    CONST robtarget p15959:= [[1433.0986274492811, 9.608746814305746, 1008.500033578516], [0, 0, 1, 0], [0, 0, 0, 0], [9E9, 9E9, 9E9, 9E9, 9E9, 9E9]];
    CONST robtarget p15960:= [[1433.1589710304575, 10.015424002704279, 1008.500033578516], [0, 0, 1, 0], [0, 0, 0, 0], [9E9, 9E9, 9E9, 9E9, 9E9, 9E9]];
    CONST robtarget p15961:= [[1433.2058201782734, 10.459822262926878, 1008.500033578516], [0, 0, 1, 0], [0, 0, 0, 0], [9E9, 9E9, 9E9, 9E9, 9E9, 9E9]];
    CONST robtarget p15962:= [[1433.4130381026719, 11.206085604370102, 1008.500033578516], [0, 0, 1, 0], [0, 0, 0, 0], [9E9, 9E9, 9E9, 9E9, 9E9, 9E9]];
    CONST robtarget p15963:= [[1433.6247056823859, 12.59383709002276, 1008.500033578516], [0, 0, 1, 0], [0, 0, 0, 0], [9E9, 9E9, 9E9, 9E9, 9E9, 9E9]];
    CONST robtarget p15964:= [[1433.6430735052686, 12.762150805315983, 1008.500033578516], [0, 0, 1, 0], [0, 0, 0, 0], [9E9, 9E9, 9E9, 9E9, 9E9, 9E9]];
    CONST robtarget p15965:= [[1433.7465034826027, 13.275407559875234, 1008.500033578516], [0, 0, 1, 0], [0, 0, 0, 0], [9E9, 9E9, 9E9, 9E9, 9E9, 9E9]];
    CONST robtarget p15966:= [[1433.7741777327235, 13.488161726566162, 1008.500033578516], [0, 0, 1, 0], [0, 0, 0, 0], [9E9, 9E9, 9E9, 9E9, 9E9, 9E9]];
    CONST robtarget p15967:= [[1433.8795125581278, 13.879378212952375, 1008.500033578516], [0, 0, 1, 0], [0, 0, 0, 0], [9E9, 9E9, 9E9, 9E9, 9E9, 9E9]];
    CONST robtarget p15968:= [[1433.9684930832368, 14.246080535111645, 1008.500033578516], [0, 0, 1, 0], [0, 0, 0, 0], [9E9, 9E9, 9E9, 9E9, 9E9, 9E9]];
    CONST robtarget p15969:= [[1434.0660993207537, 14.620211943199038, 1008.500033578516], [0, 0, 1, 0], [0, 0, 0, 0], [9E9, 9E9, 9E9, 9E9, 9E9, 9E9]];
    CONST robtarget p15970:= [[1434.095837116519, 14.758515891180053, 1008.500033578516], [0, 0, 1, 0], [0, 0, 0, 0], [9E9, 9E9, 9E9, 9E9, 9E9, 9E9]];
    CONST robtarget p15971:= [[1434.245693850769, 15.479233166590063, 1008.500033578516], [0, 0, 1, 0], [0, 0, 0, 0], [9E9, 9E9, 9E9, 9E9, 9E9, 9E9]];
    CONST robtarget p15972:= [[1434.4221561340992, 16.325849023968487, 1008.500033578516], [0, 0, 1, 0], [0, 0, 0, 0], [9E9, 9E9, 9E9, 9E9, 9E9, 9E9]];
    CONST robtarget p15973:= [[1434.61472670305, 16.937455427209215, 1008.500033578516], [0, 0, 1, 0], [0, 0, 0, 0], [9E9, 9E9, 9E9, 9E9, 9E9, 9E9]];
    CONST robtarget p15974:= [[1434.7025719249725, 17.322639850120922, 1008.500033578516], [0, 0, 1, 0], [0, 0, 0, 0], [9E9, 9E9, 9E9, 9E9, 9E9, 9E9]];
    CONST robtarget p15975:= [[1434.9090055185184, 18.0090372974757, 1008.500033578516], [0, 0, 1, 0], [0, 0, 0, 0], [9E9, 9E9, 9E9, 9E9, 9E9, 9E9]];
    CONST robtarget p15976:= [[1435.0307135396993, 18.599825888870924, 1008.500033578516], [0, 0, 1, 0], [0, 0, 0, 0], [9E9, 9E9, 9E9, 9E9, 9E9, 9E9]];
    CONST robtarget p15977:= [[1435.0769349823054, 18.84950465909236, 1008.500033578516], [0, 0, 1, 0], [0, 0, 0, 0], [9E9, 9E9, 9E9, 9E9, 9E9, 9E9]];
    CONST robtarget p15978:= [[1435.1457068870573, 19.06963509468285, 1008.500033578516], [0, 0, 1, 0], [0, 0, 0, 0], [9E9, 9E9, 9E9, 9E9, 9E9, 9E9]];
    CONST robtarget p15979:= [[1435.2539630872568, 19.45271986997699, 1008.500033578516], [0, 0, 1, 0], [0, 0, 0, 0], [9E9, 9E9, 9E9, 9E9, 9E9, 9E9]];
    CONST robtarget p15980:= [[1435.2779629825206, 19.54379334494176, 1008.500033578516], [0, 0, 1, 0], [0, 0, 0, 0], [9E9, 9E9, 9E9, 9E9, 9E9, 9E9]];
    CONST robtarget p15981:= [[1435.30275284433, 19.612075769745374, 1008.500033578516], [0, 0, 1, 0], [0, 0, 0, 0], [9E9, 9E9, 9E9, 9E9, 9E9, 9E9]];
    CONST robtarget p15982:= [[1435.4854707109937, 20.199981390981975, 1008.500033578516], [0, 0, 1, 0], [0, 0, 0, 0], [9E9, 9E9, 9E9, 9E9, 9E9, 9E9]];
    CONST robtarget p15983:= [[1435.5853392667057, 20.482104936748172, 1008.500033578516], [0, 0, 1, 0], [0, 0, 0, 0], [9E9, 9E9, 9E9, 9E9, 9E9, 9E9]];
    CONST robtarget p15984:= [[1435.7681134476982, 21.021407578977716, 1008.500033578516], [0, 0, 1, 0], [0, 0, 0, 0], [9E9, 9E9, 9E9, 9E9, 9E9, 9E9]];
    CONST robtarget p15985:= [[1435.958175713581, 21.47955589963057, 1008.500033578516], [0, 0, 1, 0], [0, 0, 0, 0], [9E9, 9E9, 9E9, 9E9, 9E9, 9E9]];
    CONST robtarget p15986:= [[1436.1023198224916, 21.945686573091862, 1008.500033578516], [0, 0, 1, 0], [0, 0, 0, 0], [9E9, 9E9, 9E9, 9E9, 9E9, 9E9]];
    CONST robtarget p15987:= [[1436.1825943607196, 22.203311510029366, 1008.500033578516], [0, 0, 1, 0], [0, 0, 0, 0], [9E9, 9E9, 9E9, 9E9, 9E9, 9E9]];
    CONST robtarget p15988:= [[1436.349538758373, 22.703386458321205, 1008.500033578516], [0, 0, 1, 0], [0, 0, 0, 0], [9E9, 9E9, 9E9, 9E9, 9E9, 9E9]];
    CONST robtarget p15989:= [[1436.6119112199715, 23.432726370190338, 1008.500033578516], [0, 0, 1, 0], [0, 0, 0, 0], [9E9, 9E9, 9E9, 9E9, 9E9, 9E9]];
    CONST robtarget p15990:= [[1436.7778943099147, 23.981953823344938, 1008.500033578516], [0, 0, 1, 0], [0, 0, 0, 0], [9E9, 9E9, 9E9, 9E9, 9E9, 9E9]];
    CONST robtarget p15991:= [[1437.0642227941967, 24.65637773782116, 1008.500033578516], [0, 0, 1, 0], [0, 0, 0, 0], [9E9, 9E9, 9E9, 9E9, 9E9, 9E9]];
    CONST robtarget p15992:= [[1437.2587373872966, 25.12385144143589, 1008.500033578516], [0, 0, 1, 0], [0, 0, 0, 0], [9E9, 9E9, 9E9, 9E9, 9E9, 9E9]];
    CONST robtarget p15993:= [[1437.3936146926897, 25.408671993782846, 1008.500033578516], [0, 0, 1, 0], [0, 0, 0, 0], [9E9, 9E9, 9E9, 9E9, 9E9, 9E9]];
    CONST robtarget p15994:= [[1437.6905856905832, 26.057288547637995, 1008.500033578516], [0, 0, 1, 0], [0, 0, 0, 0], [9E9, 9E9, 9E9, 9E9, 9E9, 9E9]];
    CONST robtarget p15995:= [[1437.8323968402112, 26.419387210097497, 1008.500033578516], [0, 0, 1, 0], [0, 0, 0, 0], [9E9, 9E9, 9E9, 9E9, 9E9, 9E9]];
    CONST robtarget p15996:= [[1437.954968895154, 26.72409400055281, 1008.500033578516], [0, 0, 1, 0], [0, 0, 0, 0], [9E9, 9E9, 9E9, 9E9, 9E9, 9E9]];
    CONST robtarget p15997:= [[1438.0143479796734, 26.878363265785197, 1008.500033578516], [0, 0, 1, 0], [0, 0, 0, 0], [9E9, 9E9, 9E9, 9E9, 9E9, 9E9]];
    CONST robtarget p15998:= [[1438.0697366851261, 27.02314795976943, 1008.500033578516], [0, 0, 1, 0], [0, 0, 0, 0], [9E9, 9E9, 9E9, 9E9, 9E9, 9E9]];
    CONST robtarget p15999:= [[1438.2271993834418, 27.43282297537347, 1008.500033578516], [0, 0, 1, 0], [0, 0, 0, 0], [9E9, 9E9, 9E9, 9E9, 9E9, 9E9]];
    CONST robtarget p16000:= [[1438.4463940522078, 27.84677822927749, 1008.500033578516], [0, 0, 1, 0], [0, 0, 0, 0], [9E9, 9E9, 9E9, 9E9, 9E9, 9E9]];
    CONST robtarget p16001:= [[1438.7558501610374, 28.663010257655827, 1008.500033578516], [0, 0, 1, 0], [0, 0, 0, 0], [9E9, 9E9, 9E9, 9E9, 9E9, 9E9]];
    CONST robtarget p16002:= [[1438.9070799315605, 28.90804462441197, 1008.500033578516], [0, 0, 1, 0], [0, 0, 0, 0], [9E9, 9E9, 9E9, 9E9, 9E9, 9E9]];
    CONST robtarget p16003:= [[1439.2433018788113, 29.59362072222892, 1008.500033578516], [0, 0, 1, 0], [0, 0, 0, 0], [9E9, 9E9, 9E9, 9E9, 9E9, 9E9]];
    CONST robtarget p16004:= [[1439.4746197403977, 30.0450442591478, 1008.500033578516], [0, 0, 1, 0], [0, 0, 0, 0], [9E9, 9E9, 9E9, 9E9, 9E9, 9E9]];
    CONST robtarget p16005:= [[1439.7668782569137, 30.57529808046486, 1008.500033578516], [0, 0, 1, 0], [0, 0, 0, 0], [9E9, 9E9, 9E9, 9E9, 9E9, 9E9]];
    CONST robtarget p16006:= [[1440.177882853498, 31.2929706114746, 1008.500033578516], [0, 0, 1, 0], [0, 0, 0, 0], [9E9, 9E9, 9E9, 9E9, 9E9, 9E9]];
    CONST robtarget p16007:= [[1440.5677510154408, 32.1772795548887, 1008.500033578516], [0, 0, 1, 0], [0, 0, 0, 0], [9E9, 9E9, 9E9, 9E9, 9E9, 9E9]];
    CONST robtarget p16008:= [[1440.9506297367848, 32.90687188456482, 1008.500033578516], [0, 0, 1, 0], [0, 0, 0, 0], [9E9, 9E9, 9E9, 9E9, 9E9, 9E9]];
    CONST robtarget p16009:= [[1441.0515934210391, 33.082825334749856, 1008.500033578516], [0, 0, 1, 0], [0, 0, 0, 0], [9E9, 9E9, 9E9, 9E9, 9E9, 9E9]];
    CONST robtarget p16010:= [[1441.291561344643, 33.51277826861488, 1008.500033578516], [0, 0, 1, 0], [0, 0, 0, 0], [9E9, 9E9, 9E9, 9E9, 9E9, 9E9]];
    CONST robtarget p16011:= [[1441.4170597081568, 33.71755199461752, 1008.500033578516], [0, 0, 1, 0], [0, 0, 0, 0], [9E9, 9E9, 9E9, 9E9, 9E9, 9E9]];
    CONST robtarget p16012:= [[1441.6717736369376, 34.087403365805486, 1008.500033578516], [0, 0, 1, 0], [0, 0, 0, 0], [9E9, 9E9, 9E9, 9E9, 9E9, 9E9]];
    CONST robtarget p16013:= [[1442.0183475741433, 34.67340426693394, 1008.500033578516], [0, 0, 1, 0], [0, 0, 0, 0], [9E9, 9E9, 9E9, 9E9, 9E9, 9E9]];
    CONST robtarget p16014:= [[1442.1305600956955, 34.842443823146525, 1008.500033578516], [0, 0, 1, 0], [0, 0, 0, 0], [9E9, 9E9, 9E9, 9E9, 9E9, 9E9]];
    CONST robtarget p16015:= [[1442.8215804591978, 35.99192933058819, 1008.500033578516], [0, 0, 1, 0], [0, 0, 0, 0], [9E9, 9E9, 9E9, 9E9, 9E9, 9E9]];
    CONST robtarget p16016:= [[1443.1406638568508, 36.489162717446646, 1008.500033578516], [0, 0, 1, 0], [0, 0, 0, 0], [9E9, 9E9, 9E9, 9E9, 9E9, 9E9]];
    CONST robtarget p16017:= [[1443.254415228456, 36.68748397793732, 1008.500033578516], [0, 0, 1, 0], [0, 0, 0, 0], [9E9, 9E9, 9E9, 9E9, 9E9, 9E9]];
    CONST robtarget p16018:= [[1443.4510665943017, 37.071600292545924, 1008.500033578516], [0, 0, 1, 0], [0, 0, 0, 0], [9E9, 9E9, 9E9, 9E9, 9E9, 9E9]];
    CONST robtarget p16019:= [[1443.9592495899064, 37.76667396099968, 1008.500033578516], [0, 0, 1, 0], [0, 0, 0, 0], [9E9, 9E9, 9E9, 9E9, 9E9, 9E9]];
    CONST robtarget p16020:= [[1444.4069080527252, 38.4188532456172, 1008.500033578516], [0, 0, 1, 0], [0, 0, 0, 0], [9E9, 9E9, 9E9, 9E9, 9E9, 9E9]];
    CONST robtarget p16021:= [[1444.7601463802437, 38.874871104904, 1008.500033578516], [0, 0, 1, 0], [0, 0, 0, 0], [9E9, 9E9, 9E9, 9E9, 9E9, 9E9]];
    CONST robtarget p16022:= [[1445.248558127412, 39.600155696272054, 1008.500033578516], [0, 0, 1, 0], [0, 0, 0, 0], [9E9, 9E9, 9E9, 9E9, 9E9, 9E9]];
    CONST robtarget p16023:= [[1445.294443015287, 39.67172478622983, 1008.500033578516], [0, 0, 1, 0], [0, 0, 0, 0], [9E9, 9E9, 9E9, 9E9, 9E9, 9E9]];
    CONST robtarget p16024:= [[1445.3797142458502, 39.77745344396661, 1008.500033578516], [0, 0, 1, 0], [0, 0, 0, 0], [9E9, 9E9, 9E9, 9E9, 9E9, 9E9]];
    CONST robtarget p16025:= [[1445.7587485571103, 40.28723104743635, 1008.500033578516], [0, 0, 1, 0], [0, 0, 0, 0], [9E9, 9E9, 9E9, 9E9, 9E9, 9E9]];
    CONST robtarget p16026:= [[1446.01804192666, 40.63892152668981, 1008.500033578516], [0, 0, 1, 0], [0, 0, 0, 0], [9E9, 9E9, 9E9, 9E9, 9E9, 9E9]];
    CONST robtarget p16027:= [[1446.312375477045, 41.03187796392518, 1008.500033578516], [0, 0, 1, 0], [0, 0, 0, 0], [9E9, 9E9, 9E9, 9E9, 9E9, 9E9]];
    CONST robtarget p16028:= [[1446.4254911527705, 41.16274682131454, 1008.500033578516], [0, 0, 1, 0], [0, 0, 0, 0], [9E9, 9E9, 9E9, 9E9, 9E9, 9E9]];
    CONST robtarget p16029:= [[1446.9971446431318, 41.842211595922834, 1008.500033578516], [0, 0, 1, 0], [0, 0, 0, 0], [9E9, 9E9, 9E9, 9E9, 9E9, 9E9]];
    CONST robtarget p16030:= [[1447.3278104158244, 42.321049762311645, 1008.500033578516], [0, 0, 1, 0], [0, 0, 0, 0], [9E9, 9E9, 9E9, 9E9, 9E9, 9E9]];
    CONST robtarget p16031:= [[1447.6388954335016, 42.65857624043116, 1008.500033578516], [0, 0, 1, 0], [0, 0, 0, 0], [9E9, 9E9, 9E9, 9E9, 9E9, 9E9]];
    CONST robtarget p16032:= [[1448.0381842833888, 43.178669383244966, 1008.500033578516], [0, 0, 1, 0], [0, 0, 0, 0], [9E9, 9E9, 9E9, 9E9, 9E9, 9E9]];
    CONST robtarget p16033:= [[1448.366752181317, 43.60401220044736, 1008.500033578516], [0, 0, 1, 0], [0, 0, 0, 0], [9E9, 9E9, 9E9, 9E9, 9E9, 9E9]];
    CONST robtarget p16034:= [[1448.5125298028045, 43.76454658599833, 1008.500033578516], [0, 0, 1, 0], [0, 0, 0, 0], [9E9, 9E9, 9E9, 9E9, 9E9, 9E9]];
    CONST robtarget p16035:= [[1448.7672952912585, 44.07132722933555, 1008.500033578516], [0, 0, 1, 0], [0, 0, 0, 0], [9E9, 9E9, 9E9, 9E9, 9E9, 9E9]];
    CONST robtarget p16036:= [[1448.8959019275212, 44.23908948956813, 1008.500033578516], [0, 0, 1, 0], [0, 0, 0, 0], [9E9, 9E9, 9E9, 9E9, 9E9, 9E9]];
    CONST robtarget p16037:= [[1449.370100010796, 44.79298202076008, 1008.500033578516], [0, 0, 1, 0], [0, 0, 0, 0], [9E9, 9E9, 9E9, 9E9, 9E9, 9E9]];
    CONST robtarget p16038:= [[1449.6542498624392, 45.13519542056041, 1008.500033578516], [0, 0, 1, 0], [0, 0, 0, 0], [9E9, 9E9, 9E9, 9E9, 9E9, 9E9]];
    CONST robtarget p16039:= [[1450.0422345772163, 45.543467221448225, 1008.500033578516], [0, 0, 1, 0], [0, 0, 0, 0], [9E9, 9E9, 9E9, 9E9, 9E9, 9E9]];
    CONST robtarget p16040:= [[1450.2040440579574, 45.71817288177934, 1008.500033578516], [0, 0, 1, 0], [0, 0, 0, 0], [9E9, 9E9, 9E9, 9E9, 9E9, 9E9]];
    CONST robtarget p16041:= [[1450.3091274651724, 45.82840814678741, 1008.500033578516], [0, 0, 1, 0], [0, 0, 0, 0], [9E9, 9E9, 9E9, 9E9, 9E9, 9E9]];
    CONST robtarget p16042:= [[1450.9473938376493, 46.4821391589785, 1008.500033578516], [0, 0, 1, 0], [0, 0, 0, 0], [9E9, 9E9, 9E9, 9E9, 9E9, 9E9]];
    CONST robtarget p16043:= [[1450.9957832882635, 46.52395188359111, 1008.500033578516], [0, 0, 1, 0], [0, 0, 0, 0], [9E9, 9E9, 9E9, 9E9, 9E9, 9E9]];
    CONST robtarget p16044:= [[1451.7155226178386, 47.278740711164716, 1008.500033578516], [0, 0, 1, 0], [0, 0, 0, 0], [9E9, 9E9, 9E9, 9E9, 9E9, 9E9]];
    CONST robtarget p16045:= [[1452.0066936624107, 47.514531408844235, 1008.500033578516], [0, 0, 1, 0], [0, 0, 0, 0], [9E9, 9E9, 9E9, 9E9, 9E9, 9E9]];
    CONST robtarget p16046:= [[1452.819568469486, 48.38961771662724, 1008.500033578516], [0, 0, 1, 0], [0, 0, 0, 0], [9E9, 9E9, 9E9, 9E9, 9E9, 9E9]];
    CONST robtarget p16047:= [[1452.9985057293763, 48.57452860134997, 1008.500033578516], [0, 0, 1, 0], [0, 0, 0, 0], [9E9, 9E9, 9E9, 9E9, 9E9, 9E9]];
    CONST robtarget p16048:= [[1453.1607314633538, 48.726012756792926, 1008.500033578516], [0, 0, 1, 0], [0, 0, 0, 0], [9E9, 9E9, 9E9, 9E9, 9E9, 9E9]];
    CONST robtarget p16049:= [[1453.7445432859734, 49.218575063884884, 1008.500033578516], [0, 0, 1, 0], [0, 0, 0, 0], [9E9, 9E9, 9E9, 9E9, 9E9, 9E9]];
    CONST robtarget p16050:= [[1454.7940861084255, 50.132860858256095, 1008.500033578516], [0, 0, 1, 0], [0, 0, 0, 0], [9E9, 9E9, 9E9, 9E9, 9E9, 9E9]];
    CONST robtarget p16051:= [[1455.1345269082879, 50.482804580104826, 1008.500033578516], [0, 0, 1, 0], [0, 0, 0, 0], [9E9, 9E9, 9E9, 9E9, 9E9, 9E9]];
    CONST robtarget p16052:= [[1455.227071666578, 50.5658550389919, 1008.500033578516], [0, 0, 1, 0], [0, 0, 0, 0], [9E9, 9E9, 9E9, 9E9, 9E9, 9E9]];
    CONST robtarget p16053:= [[1455.6269919024444, 50.9605811368297, 1008.500033578516], [0, 0, 1, 0], [0, 0, 0, 0], [9E9, 9E9, 9E9, 9E9, 9E9, 9E9]];
    CONST robtarget p16054:= [[1456.0073394176372, 51.295576906607735, 1008.500033578516], [0, 0, 1, 0], [0, 0, 0, 0], [9E9, 9E9, 9E9, 9E9, 9E9, 9E9]];
    CONST robtarget p16055:= [[1456.365165987351, 51.53794146787638, 1008.500033578516], [0, 0, 1, 0], [0, 0, 0, 0], [9E9, 9E9, 9E9, 9E9, 9E9, 9E9]];
    CONST robtarget p16056:= [[1456.7218427224004, 51.824237459893865, 1008.500033578516], [0, 0, 1, 0], [0, 0, 0, 0], [9E9, 9E9, 9E9, 9E9, 9E9, 9E9]];
    CONST robtarget p16057:= [[1457.1061071825457, 52.135035916085414, 1008.500033578516], [0, 0, 1, 0], [0, 0, 0, 0], [9E9, 9E9, 9E9, 9E9, 9E9, 9E9]];
    CONST robtarget p16058:= [[1457.31725938432, 52.3307381885903, 1008.500033578516], [0, 0, 1, 0], [0, 0, 0, 0], [9E9, 9E9, 9E9, 9E9, 9E9, 9E9]];
    CONST robtarget p16059:= [[1457.5213771439894, 52.51008271609318, 1008.500033578516], [0, 0, 1, 0], [0, 0, 0, 0], [9E9, 9E9, 9E9, 9E9, 9E9, 9E9]];
    CONST robtarget p16060:= [[1458.0058377174564, 52.939319339285575, 1008.500033578516], [0, 0, 1, 0], [0, 0, 0, 0], [9E9, 9E9, 9E9, 9E9, 9E9, 9E9]];
    CONST robtarget p16061:= [[1458.2346197754755, 53.12037415318781, 1008.500033578516], [0, 0, 1, 0], [0, 0, 0, 0], [9E9, 9E9, 9E9, 9E9, 9E9, 9E9]];
    CONST robtarget p16062:= [[1458.4753867676218, 53.31803265534384, 1008.500033578516], [0, 0, 1, 0], [0, 0, 0, 0], [9E9, 9E9, 9E9, 9E9, 9E9, 9E9]];
    CONST robtarget p16063:= [[1459.1866304764721, 53.86311971572097, 1008.500033578516], [0, 0, 1, 0], [0, 0, 0, 0], [9E9, 9E9, 9E9, 9E9, 9E9, 9E9]];
    CONST robtarget p16064:= [[1459.5783665663823, 54.16274268207515, 1008.500033578516], [0, 0, 1, 0], [0, 0, 0, 0], [9E9, 9E9, 9E9, 9E9, 9E9, 9E9]];
    CONST robtarget p16065:= [[1460.092036730576, 54.55706788749421, 1008.500033578516], [0, 0, 1, 0], [0, 0, 0, 0], [9E9, 9E9, 9E9, 9E9, 9E9, 9E9]];
    CONST robtarget p16066:= [[1460.439296844968, 54.809426933883486, 1008.500033578516], [0, 0, 1, 0], [0, 0, 0, 0], [9E9, 9E9, 9E9, 9E9, 9E9, 9E9]];
    CONST robtarget p16067:= [[1461.0793595905463, 55.18692329928378, 1008.500033578516], [0, 0, 1, 0], [0, 0, 0, 0], [9E9, 9E9, 9E9, 9E9, 9E9, 9E9]];
    CONST robtarget p16068:= [[1461.4788564955038, 55.4698326142864, 1008.500033578516], [0, 0, 1, 0], [0, 0, 0, 0], [9E9, 9E9, 9E9, 9E9, 9E9, 9E9]];
    CONST robtarget p16069:= [[1461.7693278479605, 55.68830870265511, 1008.500033578516], [0, 0, 1, 0], [0, 0, 0, 0], [9E9, 9E9, 9E9, 9E9, 9E9, 9E9]];
    CONST robtarget p16070:= [[1462.5628532139813, 56.23190731327715, 1008.500033578516], [0, 0, 1, 0], [0, 0, 0, 0], [9E9, 9E9, 9E9, 9E9, 9E9, 9E9]];
    CONST robtarget p16071:= [[1463.1232211478666, 56.58443852926386, 1008.500033578516], [0, 0, 1, 0], [0, 0, 0, 0], [9E9, 9E9, 9E9, 9E9, 9E9, 9E9]];
    CONST robtarget p16072:= [[1463.521763499162, 56.82878485469996, 1008.500033578516], [0, 0, 1, 0], [0, 0, 0, 0], [9E9, 9E9, 9E9, 9E9, 9E9, 9E9]];
    CONST robtarget p16073:= [[1463.7773127293735, 56.995022788131635, 1008.500033578516], [0, 0, 1, 0], [0, 0, 0, 0], [9E9, 9E9, 9E9, 9E9, 9E9, 9E9]];
    CONST robtarget p16074:= [[1464.4551457214025, 57.50202593561478, 1008.500033578516], [0, 0, 1, 0], [0, 0, 0, 0], [9E9, 9E9, 9E9, 9E9, 9E9, 9E9]];
    CONST robtarget p16075:= [[1464.5634203550285, 57.582022237922885, 1008.500033578516], [0, 0, 1, 0], [0, 0, 0, 0], [9E9, 9E9, 9E9, 9E9, 9E9, 9E9]];
    CONST robtarget p16076:= [[1465.3697400458088, 58.03018317718825, 1008.500033578516], [0, 0, 1, 0], [0, 0, 0, 0], [9E9, 9E9, 9E9, 9E9, 9E9, 9E9]];
    CONST robtarget p16077:= [[1465.648482730122, 58.2044987062731, 1008.500033578516], [0, 0, 1, 0], [0, 0, 0, 0], [9E9, 9E9, 9E9, 9E9, 9E9, 9E9]];
    CONST robtarget p16078:= [[1466.5459769316658, 58.67399264961996, 1008.500033578516], [0, 0, 1, 0], [0, 0, 0, 0], [9E9, 9E9, 9E9, 9E9, 9E9, 9E9]];
    CONST robtarget p16079:= [[1467.2267657129917, 59.06916037560579, 1008.500033578516], [0, 0, 1, 0], [0, 0, 0, 0], [9E9, 9E9, 9E9, 9E9, 9E9, 9E9]];
    CONST robtarget p16080:= [[1467.4882437706783, 59.24498946545437, 1008.500033578516], [0, 0, 1, 0], [0, 0, 0, 0], [9E9, 9E9, 9E9, 9E9, 9E9, 9E9]];
    CONST robtarget p16081:= [[1468.335152973493, 59.716267453443905, 1008.500033578516], [0, 0, 1, 0], [0, 0, 0, 0], [9E9, 9E9, 9E9, 9E9, 9E9, 9E9]];
    CONST robtarget p16082:= [[1468.7039832326864, 59.93135399411206, 1008.500033578516], [0, 0, 1, 0], [0, 0, 0, 0], [9E9, 9E9, 9E9, 9E9, 9E9, 9E9]];
    CONST robtarget p16083:= [[1468.9288938913592, 60.052710468605156, 1008.500033578516], [0, 0, 1, 0], [0, 0, 0, 0], [9E9, 9E9, 9E9, 9E9, 9E9, 9E9]];
    CONST robtarget p16084:= [[1469.2287228891173, 60.19182362147508, 1008.500033578516], [0, 0, 1, 0], [0, 0, 0, 0], [9E9, 9E9, 9E9, 9E9, 9E9, 9E9]];
    CONST robtarget p16085:= [[1469.6140218006096, 60.34701858277806, 1008.500033578516], [0, 0, 1, 0], [0, 0, 0, 0], [9E9, 9E9, 9E9, 9E9, 9E9, 9E9]];
    CONST robtarget p16086:= [[1470.1026517957218, 60.59639678173447, 1008.500033578516], [0, 0, 1, 0], [0, 0, 0, 0], [9E9, 9E9, 9E9, 9E9, 9E9, 9E9]];
    CONST robtarget p16087:= [[1470.2536767172498, 60.67977709489561, 1008.500033578516], [0, 0, 1, 0], [0, 0, 0, 0], [9E9, 9E9, 9E9, 9E9, 9E9, 9E9]];
    CONST robtarget p16088:= [[1470.7592636269485, 60.922434583980746, 1008.500033578516], [0, 0, 1, 0], [0, 0, 0, 0], [9E9, 9E9, 9E9, 9E9, 9E9, 9E9]];
    CONST robtarget p16089:= [[1471.4774661086992, 61.24033769839146, 1008.500033578516], [0, 0, 1, 0], [0, 0, 0, 0], [9E9, 9E9, 9E9, 9E9, 9E9, 9E9]];
    CONST robtarget p16090:= [[1471.8715766966163, 61.4248219887172, 1008.500033578516], [0, 0, 1, 0], [0, 0, 0, 0], [9E9, 9E9, 9E9, 9E9, 9E9, 9E9]];
    CONST robtarget p16091:= [[1471.9674616417628, 61.457078216292885, 1008.500033578516], [0, 0, 1, 0], [0, 0, 0, 0], [9E9, 9E9, 9E9, 9E9, 9E9, 9E9]];
    CONST robtarget p16092:= [[1472.364016831223, 61.612362344466916, 1008.500033578516], [0, 0, 1, 0], [0, 0, 0, 0], [9E9, 9E9, 9E9, 9E9, 9E9, 9E9]];
    CONST robtarget p16093:= [[1473.1130099423196, 62.020589469095526, 1008.500033578516], [0, 0, 1, 0], [0, 0, 0, 0], [9E9, 9E9, 9E9, 9E9, 9E9, 9E9]];
    CONST robtarget p16094:= [[1473.5909589644843, 62.24984289507732, 1008.500033578516], [0, 0, 1, 0], [0, 0, 0, 0], [9E9, 9E9, 9E9, 9E9, 9E9, 9E9]];
    CONST robtarget p16095:= [[1474.4024790178728, 62.50572998601946, 1008.500033578516], [0, 0, 1, 0], [0, 0, 0, 0], [9E9, 9E9, 9E9, 9E9, 9E9, 9E9]];
    CONST robtarget p16096:= [[1474.4915990041206, 62.54050880271056, 1008.500033578516], [0, 0, 1, 0], [0, 0, 0, 0], [9E9, 9E9, 9E9, 9E9, 9E9, 9E9]];
    CONST robtarget p16097:= [[1475.5468209860994, 62.99678579708994, 1008.500033578516], [0, 0, 1, 0], [0, 0, 0, 0], [9E9, 9E9, 9E9, 9E9, 9E9, 9E9]];
    CONST robtarget p16098:= [[1476.2991070939715, 63.23770336102258, 1008.500033578516], [0, 0, 1, 0], [0, 0, 0, 0], [9E9, 9E9, 9E9, 9E9, 9E9, 9E9]];
    CONST robtarget p16099:= [[1476.9969680414317, 63.53486410981911, 1008.500033578516], [0, 0, 1, 0], [0, 0, 0, 0], [9E9, 9E9, 9E9, 9E9, 9E9, 9E9]];
    CONST robtarget p16100:= [[1477.1031209594382, 63.5877638034752, 1008.500033578516], [0, 0, 1, 0], [0, 0, 0, 0], [9E9, 9E9, 9E9, 9E9, 9E9, 9E9]];
    CONST robtarget p16101:= [[1477.8877002546778, 63.89594419885661, 1008.500033578516], [0, 0, 1, 0], [0, 0, 0, 0], [9E9, 9E9, 9E9, 9E9, 9E9, 9E9]];
    CONST robtarget p16102:= [[1478.2400566872573, 64.01704825289109, 1008.500033578516], [0, 0, 1, 0], [0, 0, 0, 0], [9E9, 9E9, 9E9, 9E9, 9E9, 9E9]];
    CONST robtarget p16103:= [[1478.345994146256, 64.04712795534336, 1008.500033578516], [0, 0, 1, 0], [0, 0, 0, 0], [9E9, 9E9, 9E9, 9E9, 9E9, 9E9]];
    CONST robtarget p16104:= [[1478.7517092831447, 64.14905466791772, 1008.500033578516], [0, 0, 1, 0], [0, 0, 0, 0], [9E9, 9E9, 9E9, 9E9, 9E9, 9E9]];
    CONST robtarget p16105:= [[1478.8524086876168, 64.17558117655794, 1008.500033578516], [0, 0, 1, 0], [0, 0, 0, 0], [9E9, 9E9, 9E9, 9E9, 9E9, 9E9]];
    CONST robtarget p16106:= [[1479.718519822304, 64.46080555361299, 1008.500033578516], [0, 0, 1, 0], [0, 0, 0, 0], [9E9, 9E9, 9E9, 9E9, 9E9, 9E9]];
    CONST robtarget p16107:= [[1480.5030289274484, 64.69767934941392, 1008.500033578516], [0, 0, 1, 0], [0, 0, 0, 0], [9E9, 9E9, 9E9, 9E9, 9E9, 9E9]];
    CONST robtarget p16108:= [[1480.9110726806318, 64.81645895281174, 1008.500033578516], [0, 0, 1, 0], [0, 0, 0, 0], [9E9, 9E9, 9E9, 9E9, 9E9, 9E9]];
    CONST robtarget p16109:= [[1481.6433766032774, 65.00388321571923, 1008.500033578516], [0, 0, 1, 0], [0, 0, 0, 0], [9E9, 9E9, 9E9, 9E9, 9E9, 9E9]];
    CONST robtarget p16110:= [[1481.9905917485614, 65.12702015024472, 1008.500033578516], [0, 0, 1, 0], [0, 0, 0, 0], [9E9, 9E9, 9E9, 9E9, 9E9, 9E9]];
    CONST robtarget p16111:= [[1482.1456923586472, 65.18897033637579, 1008.500033578516], [0, 0, 1, 0], [0, 0, 0, 0], [9E9, 9E9, 9E9, 9E9, 9E9, 9E9]];
    CONST robtarget p16112:= [[1482.9004926805642, 65.39961580283652, 1008.500033578516], [0, 0, 1, 0], [0, 0, 0, 0], [9E9, 9E9, 9E9, 9E9, 9E9, 9E9]];
    CONST robtarget p16113:= [[1483.365839874073, 65.51834447481535, 1008.500033578516], [0, 0, 1, 0], [0, 0, 0, 0], [9E9, 9E9, 9E9, 9E9, 9E9, 9E9]];
    CONST robtarget p16114:= [[1483.6605705996853, 65.58222539415219, 1008.500033578516], [0, 0, 1, 0], [0, 0, 0, 0], [9E9, 9E9, 9E9, 9E9, 9E9, 9E9]];
    CONST robtarget p16115:= [[1484.5481365794053, 65.74235339856976, 1008.500033578516], [0, 0, 1, 0], [0, 0, 0, 0], [9E9, 9E9, 9E9, 9E9, 9E9, 9E9]];
    CONST robtarget p16116:= [[1484.808059584878, 65.8091029783888, 1008.500033578516], [0, 0, 1, 0], [0, 0, 0, 0], [9E9, 9E9, 9E9, 9E9, 9E9, 9E9]];
    CONST robtarget p16117:= [[1485.0631345345555, 65.8513283032221, 1008.500033578516], [0, 0, 1, 0], [0, 0, 0, 0], [9E9, 9E9, 9E9, 9E9, 9E9, 9E9]];
    CONST robtarget p16118:= [[1486.2552389920197, 66.12944847337478, 1008.500033578516], [0, 0, 1, 0], [0, 0, 0, 0], [9E9, 9E9, 9E9, 9E9, 9E9, 9E9]];
    CONST robtarget p16119:= [[1486.745913768524, 66.26623554672393, 1008.500033578516], [0, 0, 1, 0], [0, 0, 0, 0], [9E9, 9E9, 9E9, 9E9, 9E9, 9E9]];
    CONST robtarget p16120:= [[1487.4817176707566, 66.4107812271484, 1008.500033578516], [0, 0, 1, 0], [0, 0, 0, 0], [9E9, 9E9, 9E9, 9E9, 9E9, 9E9]];
    CONST robtarget p16121:= [[1487.8013138868932, 66.4636150444086, 1008.500033578516], [0, 0, 1, 0], [0, 0, 0, 0], [9E9, 9E9, 9E9, 9E9, 9E9, 9E9]];
    CONST robtarget p16122:= [[1488.0840775410525, 66.50182243595462, 1008.500033578516], [0, 0, 1, 0], [0, 0, 0, 0], [9E9, 9E9, 9E9, 9E9, 9E9, 9E9]];
    CONST robtarget p16123:= [[1489.3027826890939, 66.69076771360209, 1008.500033578516], [0, 0, 1, 0], [0, 0, 0, 0], [9E9, 9E9, 9E9, 9E9, 9E9, 9E9]];
    CONST robtarget p16124:= [[1489.7978599457865, 66.79304827252803, 1008.500033578516], [0, 0, 1, 0], [0, 0, 0, 0], [9E9, 9E9, 9E9, 9E9, 9E9, 9E9]];
    CONST robtarget p16125:= [[1490.1580174819467, 66.83051819801274, 1008.500033578516], [0, 0, 1, 0], [0, 0, 0, 0], [9E9, 9E9, 9E9, 9E9, 9E9, 9E9]];
    CONST robtarget p16126:= [[1490.6595211451563, 66.92553185056424, 1008.500033578516], [0, 0, 1, 0], [0, 0, 0, 0], [9E9, 9E9, 9E9, 9E9, 9E9, 9E9]];
    CONST robtarget p16127:= [[1490.7506060851072, 66.93781257995373, 1008.500033578516], [0, 0, 1, 0], [0, 0, 0, 0], [9E9, 9E9, 9E9, 9E9, 9E9, 9E9]];
    CONST robtarget p16128:= [[1491.7892838695197, 67.08840979982553, 1008.500033578516], [0, 0, 1, 0], [0, 0, 0, 0], [9E9, 9E9, 9E9, 9E9, 9E9, 9E9]];
    CONST robtarget p16129:= [[1492.609412010695, 67.20459844285106, 1008.500033578516], [0, 0, 1, 0], [0, 0, 0, 0], [9E9, 9E9, 9E9, 9E9, 9E9, 9E9]];
    CONST robtarget p16130:= [[1493.0973451461352, 67.21832178048781, 1008.500033578516], [0, 0, 1, 0], [0, 0, 0, 0], [9E9, 9E9, 9E9, 9E9, 9E9, 9E9]];
    CONST robtarget p16131:= [[1493.5457245082314, 67.27297021641742, 1008.500033578516], [0, 0, 1, 0], [0, 0, 0, 0], [9E9, 9E9, 9E9, 9E9, 9E9, 9E9]];
    CONST robtarget p16132:= [[1494.03034423735, 67.27558818178146, 1008.500033578516], [0, 0, 1, 0], [0, 0, 0, 0], [9E9, 9E9, 9E9, 9E9, 9E9, 9E9]];
    CONST robtarget p16133:= [[1495.0636953803023, 67.36500430040651, 1008.500033578516], [0, 0, 1, 0], [0, 0, 0, 0], [9E9, 9E9, 9E9, 9E9, 9E9, 9E9]];
    CONST robtarget p16134:= [[1495.2703995805252, 67.39760449846709, 1008.500033578516], [0, 0, 1, 0], [0, 0, 0, 0], [9E9, 9E9, 9E9, 9E9, 9E9, 9E9]];
    CONST robtarget p16135:= [[1495.7839124901182, 67.44502169230755, 1008.500033578516], [0, 0, 1, 0], [0, 0, 0, 0], [9E9, 9E9, 9E9, 9E9, 9E9, 9E9]];
    CONST robtarget p16136:= [[1496.0007086165217, 67.45991773551326, 1008.500033578516], [0, 0, 1, 0], [0, 0, 0, 0], [9E9, 9E9, 9E9, 9E9, 9E9, 9E9]];
    CONST robtarget p16137:= [[1496.7847911559047, 67.46272344024798, 1008.500033578516], [0, 0, 1, 0], [0, 0, 0, 0], [9E9, 9E9, 9E9, 9E9, 9E9, 9E9]];
    CONST robtarget p16138:= [[1497.2687498519829, 67.50360591691053, 1008.500033578516], [0, 0, 1, 0], [0, 0, 0, 0], [9E9, 9E9, 9E9, 9E9, 9E9, 9E9]];
    CONST robtarget p16139:= [[1497.5210972433517, 67.52959023107236, 1008.500033578516], [0, 0, 1, 0], [0, 0, 0, 0], [9E9, 9E9, 9E9, 9E9, 9E9, 9E9]];
    CONST robtarget p16140:= [[1497.7848772707148, 67.56287082641977, 1008.500033578516], [0, 0, 1, 0], [0, 0, 0, 0], [9E9, 9E9, 9E9, 9E9, 9E9, 9E9]];
    CONST robtarget p16141:= [[1498.1761011888134, 67.55980299430014, 1008.500033578516], [0, 0, 1, 0], [0, 0, 0, 0], [9E9, 9E9, 9E9, 9E9, 9E9, 9E9]];
    CONST robtarget p16142:= [[1498.4236953450243, 67.55697155979097, 1008.500033578516], [0, 0, 1, 0], [0, 0, 0, 0], [9E9, 9E9, 9E9, 9E9, 9E9, 9E9]];
    CONST robtarget p16143:= [[1498.9839871558106, 67.5253548343269, 1008.500033578516], [0, 0, 1, 0], [0, 0, 0, 0], [9E9, 9E9, 9E9, 9E9, 9E9, 9E9]];
    CONST robtarget p16144:= [[1499.65886843211, 67.56032717873323, 1008.500033578516], [0, 0, 1, 0], [0, 0, 0, 0], [9E9, 9E9, 9E9, 9E9, 9E9, 9E9]];
    CONST robtarget p16145:= [[1499.9462042677783, 67.56692831595988, 1008.500033578516], [0, 0, 1, 0], [0, 0, 0, 0], [9E9, 9E9, 9E9, 9E9, 9E9, 9E9]];
    CONST robtarget p16146:= [[1500.2999847909045, 67.57491158579852, 1008.500033578516], [0, 0, 1, 0], [0, 0, 0, 0], [9E9, 9E9, 9E9, 9E9, 9E9, 9E9]];
    CONST robtarget p16147:= [[1500.7492227826954, 67.54639637950622, 1008.500033578516], [0, 0, 1, 0], [0, 0, 0, 0], [9E9, 9E9, 9E9, 9E9, 9E9, 9E9]];
    CONST robtarget p16148:= [[1501.3524694849555, 67.55893763483307, 1008.500033578516], [0, 0, 1, 0], [0, 0, 0, 0], [9E9, 9E9, 9E9, 9E9, 9E9, 9E9]];
    CONST robtarget p16149:= [[1501.52595114314, 67.56553049459656, 1008.500033578516], [0, 0, 1, 0], [0, 0, 0, 0], [9E9, 9E9, 9E9, 9E9, 9E9, 9E9]];
    CONST robtarget p16150:= [[1501.7862752325475, 67.55872045451777, 1008.500033578516], [0, 0, 1, 0], [0, 0, 0, 0], [9E9, 9E9, 9E9, 9E9, 9E9, 9E9]];
    CONST robtarget p16151:= [[1502.1701800284568, 67.56646885587024, 1008.500033578516], [0, 0, 1, 0], [0, 0, 0, 0], [9E9, 9E9, 9E9, 9E9, 9E9, 9E9]];
    CONST robtarget p16152:= [[1503.3251299481256, 67.51117589101246, 1008.500033578516], [0, 0, 1, 0], [0, 0, 0, 0], [9E9, 9E9, 9E9, 9E9, 9E9, 9E9]];
    CONST robtarget p16153:= [[1504.1039683187046, 67.45169726007246, 1008.500033578516], [0, 0, 1, 0], [0, 0, 0, 0], [9E9, 9E9, 9E9, 9E9, 9E9, 9E9]];
    CONST robtarget p16154:= [[1504.5187567157118, 67.39926902339938, 1008.500033578516], [0, 0, 1, 0], [0, 0, 0, 0], [9E9, 9E9, 9E9, 9E9, 9E9, 9E9]];
    CONST robtarget p16155:= [[1504.8680529934197, 67.36426044088985, 1008.500033578516], [0, 0, 1, 0], [0, 0, 0, 0], [9E9, 9E9, 9E9, 9E9, 9E9, 9E9]];
    CONST robtarget p16156:= [[1505.8350786155258, 67.31132079236419, 1008.500033578516], [0, 0, 1, 0], [0, 0, 0, 0], [9E9, 9E9, 9E9, 9E9, 9E9, 9E9]];
    CONST robtarget p16157:= [[1506.1580751474153, 67.2839647927098, 1008.500033578516], [0, 0, 1, 0], [0, 0, 0, 0], [9E9, 9E9, 9E9, 9E9, 9E9, 9E9]];
    CONST robtarget p16158:= [[1506.8067126209448, 67.22499729243934, 1008.500033578516], [0, 0, 1, 0], [0, 0, 0, 0], [9E9, 9E9, 9E9, 9E9, 9E9, 9E9]];
    CONST robtarget p16159:= [[1506.914620863095, 67.22039283299013, 1008.500033578516], [0, 0, 1, 0], [0, 0, 0, 0], [9E9, 9E9, 9E9, 9E9, 9E9, 9E9]];
    CONST robtarget p16160:= [[1507.3311742469302, 67.20517243265284, 1008.500033578516], [0, 0, 1, 0], [0, 0, 0, 0], [9E9, 9E9, 9E9, 9E9, 9E9, 9E9]];
    CONST robtarget p16161:= [[1508.051846757844, 67.09798746857994, 1008.500033578516], [0, 0, 1, 0], [0, 0, 0, 0], [9E9, 9E9, 9E9, 9E9, 9E9, 9E9]];
    CONST robtarget p16162:= [[1508.4962840792496, 67.03555884808507, 1008.500033578516], [0, 0, 1, 0], [0, 0, 0, 0], [9E9, 9E9, 9E9, 9E9, 9E9, 9E9]];
    CONST robtarget p16163:= [[1508.663017896194, 67.01737314745735, 1008.500033578516], [0, 0, 1, 0], [0, 0, 0, 0], [9E9, 9E9, 9E9, 9E9, 9E9, 9E9]];
    CONST robtarget p16164:= [[1509.2280584400226, 66.92517621660978, 1008.500033578516], [0, 0, 1, 0], [0, 0, 0, 0], [9E9, 9E9, 9E9, 9E9, 9E9, 9E9]];
    CONST robtarget p16165:= [[1509.522811564534, 66.88786463160581, 1008.500033578516], [0, 0, 1, 0], [0, 0, 0, 0], [9E9, 9E9, 9E9, 9E9, 9E9, 9E9]];
    CONST robtarget p16166:= [[1510.2013580087432, 66.77658475896071, 1008.500033578516], [0, 0, 1, 0], [0, 0, 0, 0], [9E9, 9E9, 9E9, 9E9, 9E9, 9E9]];
    CONST robtarget p16167:= [[1510.861765913483, 66.67830591520884, 1008.500033578516], [0, 0, 1, 0], [0, 0, 0, 0], [9E9, 9E9, 9E9, 9E9, 9E9, 9E9]];
    CONST robtarget p16168:= [[1511.2000364271769, 66.62198389585312, 1008.500033578516], [0, 0, 1, 0], [0, 0, 0, 0], [9E9, 9E9, 9E9, 9E9, 9E9, 9E9]];
    CONST robtarget p16169:= [[1511.256665370911, 66.6101649925936, 1008.500033578516], [0, 0, 1, 0], [0, 0, 0, 0], [9E9, 9E9, 9E9, 9E9, 9E9, 9E9]];
    CONST robtarget p16170:= [[1511.6672809390207, 66.5435997052037, 1008.500033578516], [0, 0, 1, 0], [0, 0, 0, 0], [9E9, 9E9, 9E9, 9E9, 9E9, 9E9]];
    CONST robtarget p16171:= [[1512.0057148899998, 66.50992114851671, 1008.500033578516], [0, 0, 1, 0], [0, 0, 0, 0], [9E9, 9E9, 9E9, 9E9, 9E9, 9E9]];
    CONST robtarget p16172:= [[1512.242060924263, 66.4896230026395, 1008.500033578516], [0, 0, 1, 0], [0, 0, 0, 0], [9E9, 9E9, 9E9, 9E9, 9E9, 9E9]];
    CONST robtarget p16173:= [[1512.6062895353741, 66.39183579555883, 1008.500033578516], [0, 0, 1, 0], [0, 0, 0, 0], [9E9, 9E9, 9E9, 9E9, 9E9, 9E9]];
    CONST robtarget p16174:= [[1512.8154231901442, 66.33315781927045, 1008.500033578516], [0, 0, 1, 0], [0, 0, 0, 0], [9E9, 9E9, 9E9, 9E9, 9E9, 9E9]];
    CONST robtarget p16175:= [[1513.5873541229998, 66.18668536447795, 1008.500033578516], [0, 0, 1, 0], [0, 0, 0, 0], [9E9, 9E9, 9E9, 9E9, 9E9, 9E9]];
    CONST robtarget p16176:= [[1514.1141486168747, 66.07432584393821, 1008.500033578516], [0, 0, 1, 0], [0, 0, 0, 0], [9E9, 9E9, 9E9, 9E9, 9E9, 9E9]];
    CONST robtarget p16177:= [[1515.3196760163135, 65.77095272586276, 1008.500033578516], [0, 0, 1, 0], [0, 0, 0, 0], [9E9, 9E9, 9E9, 9E9, 9E9, 9E9]];
    CONST robtarget p16178:= [[1515.8977747972394, 65.67558118808309, 1008.500033578516], [0, 0, 1, 0], [0, 0, 0, 0], [9E9, 9E9, 9E9, 9E9, 9E9, 9E9]];
    CONST robtarget p16179:= [[1516.529099539786, 65.53055285760634, 1008.500033578516], [0, 0, 1, 0], [0, 0, 0, 0], [9E9, 9E9, 9E9, 9E9, 9E9, 9E9]];
    CONST robtarget p16180:= [[1516.8811698775148, 65.43150387512146, 1008.500033578516], [0, 0, 1, 0], [0, 0, 0, 0], [9E9, 9E9, 9E9, 9E9, 9E9, 9E9]];
    CONST robtarget p16181:= [[1517.2882579663342, 65.33220692496353, 1008.500033578516], [0, 0, 1, 0], [0, 0, 0, 0], [9E9, 9E9, 9E9, 9E9, 9E9, 9E9]];
    CONST robtarget p16182:= [[1517.3489242665862, 65.3183621528987, 1008.500033578516], [0, 0, 1, 0], [0, 0, 0, 0], [9E9, 9E9, 9E9, 9E9, 9E9, 9E9]];
    CONST robtarget p16183:= [[1518.0070267032497, 65.1083562925629, 1008.500033578516], [0, 0, 1, 0], [0, 0, 0, 0], [9E9, 9E9, 9E9, 9E9, 9E9, 9E9]];
    CONST robtarget p16184:= [[1518.2343526620655, 65.05429995971399, 1008.500033578516], [0, 0, 1, 0], [0, 0, 0, 0], [9E9, 9E9, 9E9, 9E9, 9E9, 9E9]];
    CONST robtarget p16185:= [[1519.1723039191336, 64.79471174169457, 1008.500033578516], [0, 0, 1, 0], [0, 0, 0, 0], [9E9, 9E9, 9E9, 9E9, 9E9, 9E9]];
    CONST robtarget p16186:= [[1519.8619834830579, 64.54927590595203, 1008.500033578516], [0, 0, 1, 0], [0, 0, 0, 0], [9E9, 9E9, 9E9, 9E9, 9E9, 9E9]];
    CONST robtarget p16187:= [[1520.4954780542823, 64.37834296249353, 1008.500033578516], [0, 0, 1, 0], [0, 0, 0, 0], [9E9, 9E9, 9E9, 9E9, 9E9, 9E9]];
    CONST robtarget p16188:= [[1520.6920151495815, 64.3358817612032, 1008.500033578516], [0, 0, 1, 0], [0, 0, 0, 0], [9E9, 9E9, 9E9, 9E9, 9E9, 9E9]];
    CONST robtarget p16189:= [[1521.0901400841094, 64.21270182988847, 1008.500033578516], [0, 0, 1, 0], [0, 0, 0, 0], [9E9, 9E9, 9E9, 9E9, 9E9, 9E9]];
    CONST robtarget p16190:= [[1521.6572040310643, 64.01071740259904, 1008.500033578516], [0, 0, 1, 0], [0, 0, 0, 0], [9E9, 9E9, 9E9, 9E9, 9E9, 9E9]];
    CONST robtarget p16191:= [[1522.4562553248777, 63.75858606397445, 1008.500033578516], [0, 0, 1, 0], [0, 0, 0, 0], [9E9, 9E9, 9E9, 9E9, 9E9, 9E9]];
    CONST robtarget p16192:= [[1522.741064368704, 63.641331237073345, 1008.500033578516], [0, 0, 1, 0], [0, 0, 0, 0], [9E9, 9E9, 9E9, 9E9, 9E9, 9E9]];
    CONST robtarget p16193:= [[1523.579829670514, 63.32728873619162, 1008.500033578516], [0, 0, 1, 0], [0, 0, 0, 0], [9E9, 9E9, 9E9, 9E9, 9E9, 9E9]];
    CONST robtarget p16194:= [[1523.6679239624505, 63.29141898338641, 1008.500033578516], [0, 0, 1, 0], [0, 0, 0, 0], [9E9, 9E9, 9E9, 9E9, 9E9, 9E9]];
    CONST robtarget p16195:= [[1524.0807512058723, 63.137895512951744, 1008.500033578516], [0, 0, 1, 0], [0, 0, 0, 0], [9E9, 9E9, 9E9, 9E9, 9E9, 9E9]];
    CONST robtarget p16196:= [[1524.991654114887, 62.77697253972876, 1008.500033578516], [0, 0, 1, 0], [0, 0, 0, 0], [9E9, 9E9, 9E9, 9E9, 9E9, 9E9]];
    CONST robtarget p16197:= [[1525.3261931070772, 62.647846139703475, 1008.500033578516], [0, 0, 1, 0], [0, 0, 0, 0], [9E9, 9E9, 9E9, 9E9, 9E9, 9E9]];
    CONST robtarget p16198:= [[1525.601768832265, 62.53814789177544, 1008.500033578516], [0, 0, 1, 0], [0, 0, 0, 0], [9E9, 9E9, 9E9, 9E9, 9E9, 9E9]];
    CONST robtarget p16199:= [[1526.0125706485137, 62.350267428342605, 1008.500033578516], [0, 0, 1, 0], [0, 0, 0, 0], [9E9, 9E9, 9E9, 9E9, 9E9, 9E9]];
    CONST robtarget p16200:= [[1526.3066542769623, 62.222073413733355, 1008.500033578516], [0, 0, 1, 0], [0, 0, 0, 0], [9E9, 9E9, 9E9, 9E9, 9E9, 9E9]];
    CONST robtarget p16201:= [[1526.5847268679495, 62.10671053591453, 1008.500033578516], [0, 0, 1, 0], [0, 0, 0, 0], [9E9, 9E9, 9E9, 9E9, 9E9, 9E9]];
    CONST robtarget p16202:= [[1527.2352319250879, 61.840380671867834, 1008.500033578516], [0, 0, 1, 0], [0, 0, 0, 0], [9E9, 9E9, 9E9, 9E9, 9E9, 9E9]];
    CONST robtarget p16203:= [[1527.7455310348773, 61.61730831770738, 1008.500033578516], [0, 0, 1, 0], [0, 0, 0, 0], [9E9, 9E9, 9E9, 9E9, 9E9, 9E9]];
    CONST robtarget p16204:= [[1528.1664657308856, 61.41094787108726, 1008.500033578516], [0, 0, 1, 0], [0, 0, 0, 0], [9E9, 9E9, 9E9, 9E9, 9E9, 9E9]];
    CONST robtarget p16205:= [[1528.9780169909725, 61.03104339091895, 1008.500033578516], [0, 0, 1, 0], [0, 0, 0, 0], [9E9, 9E9, 9E9, 9E9, 9E9, 9E9]];
    CONST robtarget p16206:= [[1529.3016355180364, 60.88030629947495, 1008.500033578516], [0, 0, 1, 0], [0, 0, 0, 0], [9E9, 9E9, 9E9, 9E9, 9E9, 9E9]];
    CONST robtarget p16207:= [[1529.6925056554678, 60.699304831064, 1008.500033578516], [0, 0, 1, 0], [0, 0, 0, 0], [9E9, 9E9, 9E9, 9E9, 9E9, 9E9]];
    CONST robtarget p16208:= [[1529.8495799186976, 60.61488918156924, 1008.500033578516], [0, 0, 1, 0], [0, 0, 0, 0], [9E9, 9E9, 9E9, 9E9, 9E9, 9E9]];
    CONST robtarget p16209:= [[1530.9252244029178, 60.13040037803857, 1008.500033578516], [0, 0, 1, 0], [0, 0, 0, 0], [9E9, 9E9, 9E9, 9E9, 9E9, 9E9]];
    CONST robtarget p16210:= [[1531.1133808775767, 60.0095698694973, 1008.500033578516], [0, 0, 1, 0], [0, 0, 0, 0], [9E9, 9E9, 9E9, 9E9, 9E9, 9E9]];
    CONST robtarget p16211:= [[1531.338252726174, 59.87470420482346, 1008.500033578516], [0, 0, 1, 0], [0, 0, 0, 0], [9E9, 9E9, 9E9, 9E9, 9E9, 9E9]];
    CONST robtarget p16212:= [[1532.6051035607525, 59.181744440511025, 1008.500033578516], [0, 0, 1, 0], [0, 0, 0, 0], [9E9, 9E9, 9E9, 9E9, 9E9, 9E9]];
    CONST robtarget p16213:= [[1532.9350906622394, 58.98976458283032, 1008.500033578516], [0, 0, 1, 0], [0, 0, 0, 0], [9E9, 9E9, 9E9, 9E9, 9E9, 9E9]];
    CONST robtarget p16214:= [[1533.539947108557, 58.6350239582536, 1008.500033578516], [0, 0, 1, 0], [0, 0, 0, 0], [9E9, 9E9, 9E9, 9E9, 9E9, 9E9]];
    CONST robtarget p16215:= [[1533.665581038032, 58.57039735642364, 1008.500033578516], [0, 0, 1, 0], [0, 0, 0, 0], [9E9, 9E9, 9E9, 9E9, 9E9, 9E9]];
    CONST robtarget p16216:= [[1533.765204579849, 58.514108898550674, 1008.500033578516], [0, 0, 1, 0], [0, 0, 0, 0], [9E9, 9E9, 9E9, 9E9, 9E9, 9E9]];
    CONST robtarget p16217:= [[1534.434498778867, 58.13371042770375, 1008.500033578516], [0, 0, 1, 0], [0, 0, 0, 0], [9E9, 9E9, 9E9, 9E9, 9E9, 9E9]];
    CONST robtarget p16218:= [[1535.0274474561854, 57.78598546325415, 1008.500033578516], [0, 0, 1, 0], [0, 0, 0, 0], [9E9, 9E9, 9E9, 9E9, 9E9, 9E9]];
    CONST robtarget p16219:= [[1535.2366628819493, 57.68664135704496, 1008.500033578516], [0, 0, 1, 0], [0, 0, 0, 0], [9E9, 9E9, 9E9, 9E9, 9E9, 9E9]];
    CONST robtarget p16220:= [[1536.2809482582015, 56.95240582097918, 1008.500033578516], [0, 0, 1, 0], [0, 0, 0, 0], [9E9, 9E9, 9E9, 9E9, 9E9, 9E9]];
    CONST robtarget p16221:= [[1536.5358434102075, 56.82379129320849, 1008.500033578516], [0, 0, 1, 0], [0, 0, 0, 0], [9E9, 9E9, 9E9, 9E9, 9E9, 9E9]];
    CONST robtarget p16222:= [[1536.7615401066853, 56.698549823481244, 1008.500033578516], [0, 0, 1, 0], [0, 0, 0, 0], [9E9, 9E9, 9E9, 9E9, 9E9, 9E9]];
    CONST robtarget p16223:= [[1537.4709825533946, 56.15506886151951, 1008.500033578516], [0, 0, 1, 0], [0, 0, 0, 0], [9E9, 9E9, 9E9, 9E9, 9E9, 9E9]];
    CONST robtarget p16224:= [[1538.14340455985, 55.70807589276281, 1008.500033578516], [0, 0, 1, 0], [0, 0, 0, 0], [9E9, 9E9, 9E9, 9E9, 9E9, 9E9]];
    CONST robtarget p16225:= [[1538.690509725695, 55.405104289167724, 1008.500033578516], [0, 0, 1, 0], [0, 0, 0, 0], [9E9, 9E9, 9E9, 9E9, 9E9, 9E9]];
    CONST robtarget p16226:= [[1539.251905817547, 54.98821800634306, 1008.500033578516], [0, 0, 1, 0], [0, 0, 0, 0], [9E9, 9E9, 9E9, 9E9, 9E9, 9E9]];
    CONST robtarget p16227:= [[1539.3888053754263, 54.896561256571744, 1008.500033578516], [0, 0, 1, 0], [0, 0, 0, 0], [9E9, 9E9, 9E9, 9E9, 9E9, 9E9]];
    CONST robtarget p16228:= [[1539.5312702958397, 54.800078078137915, 1008.500033578516], [0, 0, 1, 0], [0, 0, 0, 0], [9E9, 9E9, 9E9, 9E9, 9E9, 9E9]];
    CONST robtarget p16229:= [[1539.873034811547, 54.573144924912185, 1008.500033578516], [0, 0, 1, 0], [0, 0, 0, 0], [9E9, 9E9, 9E9, 9E9, 9E9, 9E9]];
    CONST robtarget p16230:= [[1540.4571828498044, 54.11907380497992, 1008.500033578516], [0, 0, 1, 0], [0, 0, 0, 0], [9E9, 9E9, 9E9, 9E9, 9E9, 9E9]];
    CONST robtarget p16231:= [[1540.6454968093467, 53.97304272734445, 1008.500033578516], [0, 0, 1, 0], [0, 0, 0, 0], [9E9, 9E9, 9E9, 9E9, 9E9, 9E9]];
    CONST robtarget p16232:= [[1540.8487928799423, 53.801382146093005, 1008.500033578516], [0, 0, 1, 0], [0, 0, 0, 0], [9E9, 9E9, 9E9, 9E9, 9E9, 9E9]];
    CONST robtarget p16233:= [[1541.5968777060616, 53.21746344878743, 1008.500033578516], [0, 0, 1, 0], [0, 0, 0, 0], [9E9, 9E9, 9E9, 9E9, 9E9, 9E9]];
    CONST robtarget p16234:= [[1542.1557567184345, 52.80360707323666, 1008.500033578516], [0, 0, 1, 0], [0, 0, 0, 0], [9E9, 9E9, 9E9, 9E9, 9E9, 9E9]];
    CONST robtarget p16235:= [[1542.3672580179314, 52.657895721498704, 1008.500033578516], [0, 0, 1, 0], [0, 0, 0, 0], [9E9, 9E9, 9E9, 9E9, 9E9, 9E9]];
    CONST robtarget p16236:= [[1543.1264456746446, 52.0560909500626, 1008.500033578516], [0, 0, 1, 0], [0, 0, 0, 0], [9E9, 9E9, 9E9, 9E9, 9E9, 9E9]];
    CONST robtarget p16237:= [[1543.4511631739797, 51.7464949296357, 1008.500033578516], [0, 0, 1, 0], [0, 0, 0, 0], [9E9, 9E9, 9E9, 9E9, 9E9, 9E9]];
    CONST robtarget p16238:= [[1543.7980368344502, 51.41813954769735, 1008.500033578516], [0, 0, 1, 0], [0, 0, 0, 0], [9E9, 9E9, 9E9, 9E9, 9E9, 9E9]];
    CONST robtarget p16239:= [[1544.1528809601373, 51.10559622632208, 1008.500033578516], [0, 0, 1, 0], [0, 0, 0, 0], [9E9, 9E9, 9E9, 9E9, 9E9, 9E9]];
    CONST robtarget p16240:= [[1544.632473742973, 50.7115438681728, 1008.500033578516], [0, 0, 1, 0], [0, 0, 0, 0], [9E9, 9E9, 9E9, 9E9, 9E9, 9E9]];
    CONST robtarget p16241:= [[1545.067336188595, 50.31881299810297, 1008.500033578516], [0, 0, 1, 0], [0, 0, 0, 0], [9E9, 9E9, 9E9, 9E9, 9E9, 9E9]];
    CONST robtarget p16242:= [[1545.169738603748, 50.2226523829372, 1008.500033578516], [0, 0, 1, 0], [0, 0, 0, 0], [9E9, 9E9, 9E9, 9E9, 9E9, 9E9]];
    CONST robtarget p16243:= [[1545.2203270913708, 50.17221469994723, 1008.500033578516], [0, 0, 1, 0], [0, 0, 0, 0], [9E9, 9E9, 9E9, 9E9, 9E9, 9E9]];
    CONST robtarget p16244:= [[1545.6241471030944, 49.789102055881884, 1008.500033578516], [0, 0, 1, 0], [0, 0, 0, 0], [9E9, 9E9, 9E9, 9E9, 9E9, 9E9]];
    CONST robtarget p16245:= [[1545.7969761952904, 49.63364123708452, 1008.500033578516], [0, 0, 1, 0], [0, 0, 0, 0], [9E9, 9E9, 9E9, 9E9, 9E9, 9E9]];
    CONST robtarget p16246:= [[1546.9567035638051, 48.64037268309886, 1008.500033578516], [0, 0, 1, 0], [0, 0, 0, 0], [9E9, 9E9, 9E9, 9E9, 9E9, 9E9]];
    CONST robtarget p16247:= [[1547.1137387530064, 48.48792866633548, 1008.500033578516], [0, 0, 1, 0], [0, 0, 0, 0], [9E9, 9E9, 9E9, 9E9, 9E9, 9E9]];
    CONST robtarget p16248:= [[1547.3908771598938, 48.167872617564456, 1008.500033578516], [0, 0, 1, 0], [0, 0, 0, 0], [9E9, 9E9, 9E9, 9E9, 9E9, 9E9]];
    CONST robtarget p16249:= [[1547.9286940513095, 47.63881835014034, 1008.500033578516], [0, 0, 1, 0], [0, 0, 0, 0], [9E9, 9E9, 9E9, 9E9, 9E9, 9E9]];
    CONST robtarget p16250:= [[1548.9027235955841, 46.58641968968692, 1008.500033578516], [0, 0, 1, 0], [0, 0, 0, 0], [9E9, 9E9, 9E9, 9E9, 9E9, 9E9]];
    CONST robtarget p16251:= [[1549.5994430223811, 45.91067623661789, 1008.500033578516], [0, 0, 1, 0], [0, 0, 0, 0], [9E9, 9E9, 9E9, 9E9, 9E9, 9E9]];
    CONST robtarget p16252:= [[1549.9531790001015, 45.538592434007256, 1008.500033578516], [0, 0, 1, 0], [0, 0, 0, 0], [9E9, 9E9, 9E9, 9E9, 9E9, 9E9]];
    CONST robtarget p16253:= [[1550.0864950563696, 45.38338897314145, 1008.500033578516], [0, 0, 1, 0], [0, 0, 0, 0], [9E9, 9E9, 9E9, 9E9, 9E9, 9E9]];
    CONST robtarget p16254:= [[1550.3867530528216, 45.0653065456608, 1008.500033578516], [0, 0, 1, 0], [0, 0, 0, 0], [9E9, 9E9, 9E9, 9E9, 9E9, 9E9]];
    CONST robtarget p16255:= [[1550.5252376844503, 44.90894853342681, 1008.500033578516], [0, 0, 1, 0], [0, 0, 0, 0], [9E9, 9E9, 9E9, 9E9, 9E9, 9E9]];
    CONST robtarget p16256:= [[1551.3702462240315, 43.87782235580386, 1008.500033578516], [0, 0, 1, 0], [0, 0, 0, 0], [9E9, 9E9, 9E9, 9E9, 9E9, 9E9]];
    CONST robtarget p16257:= [[1551.5306802812183, 43.711757725309965, 1008.500033578516], [0, 0, 1, 0], [0, 0, 0, 0], [9E9, 9E9, 9E9, 9E9, 9E9, 9E9]];
    CONST robtarget p16258:= [[1551.6895740014172, 43.51981024746627, 1008.500033578516], [0, 0, 1, 0], [0, 0, 0, 0], [9E9, 9E9, 9E9, 9E9, 9E9, 9E9]];
    CONST robtarget p16259:= [[1551.9241438094352, 43.227008008838794, 1008.500033578516], [0, 0, 1, 0], [0, 0, 0, 0], [9E9, 9E9, 9E9, 9E9, 9E9, 9E9]];
    CONST robtarget p16260:= [[1552.3155403705046, 42.72597601818619, 1008.500033578516], [0, 0, 1, 0], [0, 0, 0, 0], [9E9, 9E9, 9E9, 9E9, 9E9, 9E9]];
    CONST robtarget p16261:= [[1552.8155267755592, 42.16004986176419, 1008.500033578516], [0, 0, 1, 0], [0, 0, 0, 0], [9E9, 9E9, 9E9, 9E9, 9E9, 9E9]];
    CONST robtarget p16262:= [[1553.040888905037, 41.83955435388586, 1008.500033578516], [0, 0, 1, 0], [0, 0, 0, 0], [9E9, 9E9, 9E9, 9E9, 9E9, 9E9]];
    CONST robtarget p16263:= [[1553.6366244962283, 41.12032876641041, 1008.500033578516], [0, 0, 1, 0], [0, 0, 0, 0], [9E9, 9E9, 9E9, 9E9, 9E9, 9E9]];
    CONST robtarget p16264:= [[1554.0622483775878, 40.544990601836375, 1008.500033578516], [0, 0, 1, 0], [0, 0, 0, 0], [9E9, 9E9, 9E9, 9E9, 9E9, 9E9]];
    CONST robtarget p16265:= [[1554.482126760209, 39.964334016060945, 1008.500033578516], [0, 0, 1, 0], [0, 0, 0, 0], [9E9, 9E9, 9E9, 9E9, 9E9, 9E9]];
    CONST robtarget p16266:= [[1554.7876823798358, 39.51873010635322, 1008.500033578516], [0, 0, 1, 0], [0, 0, 0, 0], [9E9, 9E9, 9E9, 9E9, 9E9, 9E9]];
    CONST robtarget p16267:= [[1555.190994619107, 38.96882711559114, 1008.500033578516], [0, 0, 1, 0], [0, 0, 0, 0], [9E9, 9E9, 9E9, 9E9, 9E9, 9E9]];
    CONST robtarget p16268:= [[1555.5357512043624, 38.506678408790265, 1008.500033578516], [0, 0, 1, 0], [0, 0, 0, 0], [9E9, 9E9, 9E9, 9E9, 9E9, 9E9]];
    CONST robtarget p16269:= [[1555.654198573368, 38.338015815783976, 1008.500033578516], [0, 0, 1, 0], [0, 0, 0, 0], [9E9, 9E9, 9E9, 9E9, 9E9, 9E9]];
    CONST robtarget p16270:= [[1556.015020468224, 37.81320593308459, 1008.500033578516], [0, 0, 1, 0], [0, 0, 0, 0], [9E9, 9E9, 9E9, 9E9, 9E9, 9E9]];
    CONST robtarget p16271:= [[1556.2529437145502, 37.49349759459254, 1008.500033578516], [0, 0, 1, 0], [0, 0, 0, 0], [9E9, 9E9, 9E9, 9E9, 9E9, 9E9]];
    CONST robtarget p16272:= [[1556.3981689585596, 37.29093802411656, 1008.500033578516], [0, 0, 1, 0], [0, 0, 0, 0], [9E9, 9E9, 9E9, 9E9, 9E9, 9E9]];
    CONST robtarget p16273:= [[1556.8224023011526, 36.56324052702395, 1008.500033578516], [0, 0, 1, 0], [0, 0, 0, 0], [9E9, 9E9, 9E9, 9E9, 9E9, 9E9]];
    CONST robtarget p16274:= [[1557.0592298176236, 36.19739545688475, 1008.500033578516], [0, 0, 1, 0], [0, 0, 0, 0], [9E9, 9E9, 9E9, 9E9, 9E9, 9E9]];
    CONST robtarget p16275:= [[1557.25601028899, 35.887958184624694, 1008.500033578516], [0, 0, 1, 0], [0, 0, 0, 0], [9E9, 9E9, 9E9, 9E9, 9E9, 9E9]];
    CONST robtarget p16276:= [[1557.4357989455061, 35.550940652576685, 1008.500033578516], [0, 0, 1, 0], [0, 0, 0, 0], [9E9, 9E9, 9E9, 9E9, 9E9, 9E9]];
    CONST robtarget p16277:= [[1557.8256919941164, 34.93346399106704, 1008.500033578516], [0, 0, 1, 0], [0, 0, 0, 0], [9E9, 9E9, 9E9, 9E9, 9E9, 9E9]];
    CONST robtarget p16278:= [[1558.0786409233476, 34.539546040927036, 1008.500033578516], [0, 0, 1, 0], [0, 0, 0, 0], [9E9, 9E9, 9E9, 9E9, 9E9, 9E9]];
    CONST robtarget p16279:= [[1558.5494520993752, 33.738990861255246, 1008.500033578516], [0, 0, 1, 0], [0, 0, 0, 0], [9E9, 9E9, 9E9, 9E9, 9E9, 9E9]];
    CONST robtarget p16280:= [[1558.6677237334652, 33.554065226060175, 1008.500033578516], [0, 0, 1, 0], [0, 0, 0, 0], [9E9, 9E9, 9E9, 9E9, 9E9, 9E9]];
    CONST robtarget p16281:= [[1558.9141754255486, 33.15925656435246, 1008.500033578516], [0, 0, 1, 0], [0, 0, 0, 0], [9E9, 9E9, 9E9, 9E9, 9E9, 9E9]];
    CONST robtarget p16282:= [[1559.4219381001647, 32.15420514313904, 1008.500033578516], [0, 0, 1, 0], [0, 0, 0, 0], [9E9, 9E9, 9E9, 9E9, 9E9, 9E9]];
    CONST robtarget p16283:= [[1559.5672080614372, 31.828022421802174, 1008.500033578516], [0, 0, 1, 0], [0, 0, 0, 0], [9E9, 9E9, 9E9, 9E9, 9E9, 9E9]];
    CONST robtarget p16284:= [[1559.8201048250467, 31.36696348396636, 1008.500033578516], [0, 0, 1, 0], [0, 0, 0, 0], [9E9, 9E9, 9E9, 9E9, 9E9, 9E9]];
    CONST robtarget p16285:= [[1560.4198232136341, 30.23749965855359, 1008.500033578516], [0, 0, 1, 0], [0, 0, 0, 0], [9E9, 9E9, 9E9, 9E9, 9E9, 9E9]];
    CONST robtarget p16286:= [[1560.5058733413384, 30.081565327726125, 1008.500033578516], [0, 0, 1, 0], [0, 0, 0, 0], [9E9, 9E9, 9E9, 9E9, 9E9, 9E9]];
    CONST robtarget p16287:= [[1560.7107086566648, 29.68346384777989, 1008.500033578516], [0, 0, 1, 0], [0, 0, 0, 0], [9E9, 9E9, 9E9, 9E9, 9E9, 9E9]];
    CONST robtarget p16288:= [[1560.8006054071427, 29.503205244977394, 1008.500033578516], [0, 0, 1, 0], [0, 0, 0, 0], [9E9, 9E9, 9E9, 9E9, 9E9, 9E9]];
    CONST robtarget p16289:= [[1561.0016624643956, 29.01438936729346, 1008.500033578516], [0, 0, 1, 0], [0, 0, 0, 0], [9E9, 9E9, 9E9, 9E9, 9E9, 9E9]];
    CONST robtarget p16290:= [[1561.322585734127, 28.431959031194367, 1008.500033578516], [0, 0, 1, 0], [0, 0, 0, 0], [9E9, 9E9, 9E9, 9E9, 9E9, 9E9]];
    CONST robtarget p16291:= [[1561.6840266460151, 27.586172939296944, 1008.500033578516], [0, 0, 1, 0], [0, 0, 0, 0], [9E9, 9E9, 9E9, 9E9, 9E9, 9E9]];
    CONST robtarget p16292:= [[1561.7614330188878, 27.411241673664662, 1008.500033578516], [0, 0, 1, 0], [0, 0, 0, 0], [9E9, 9E9, 9E9, 9E9, 9E9, 9E9]];
    CONST robtarget p16293:= [[1561.8319623549032, 27.22730118404087, 1008.500033578516], [0, 0, 1, 0], [0, 0, 0, 0], [9E9, 9E9, 9E9, 9E9, 9E9, 9E9]];
    CONST robtarget p16294:= [[1562.0348298300441, 26.764763417680882, 1008.500033578516], [0, 0, 1, 0], [0, 0, 0, 0], [9E9, 9E9, 9E9, 9E9, 9E9, 9E9]];
    CONST robtarget p16295:= [[1562.113758626317, 26.578533392523056, 1008.500033578516], [0, 0, 1, 0], [0, 0, 0, 0], [9E9, 9E9, 9E9, 9E9, 9E9, 9E9]];
    CONST robtarget p16296:= [[1562.5153619602972, 25.633228337836854, 1008.500033578516], [0, 0, 1, 0], [0, 0, 0, 0], [9E9, 9E9, 9E9, 9E9, 9E9, 9E9]];
    CONST robtarget p16297:= [[1562.6404314619315, 25.331756088136615, 1008.500033578516], [0, 0, 1, 0], [0, 0, 0, 0], [9E9, 9E9, 9E9, 9E9, 9E9, 9E9]];
    CONST robtarget p16298:= [[1562.9493904188116, 24.627221500377047, 1008.500033578516], [0, 0, 1, 0], [0, 0, 0, 0], [9E9, 9E9, 9E9, 9E9, 9E9, 9E9]];
    CONST robtarget p16299:= [[1562.9600893934594, 24.60458742551745, 1008.500033578516], [0, 0, 1, 0], [0, 0, 0, 0], [9E9, 9E9, 9E9, 9E9, 9E9, 9E9]];
    CONST robtarget p16300:= [[1563.1976095893567, 23.88689186993514, 1008.500033578516], [0, 0, 1, 0], [0, 0, 0, 0], [9E9, 9E9, 9E9, 9E9, 9E9, 9E9]];
    CONST robtarget p16301:= [[1563.3135927604592, 23.59812151587404, 1008.500033578516], [0, 0, 1, 0], [0, 0, 0, 0], [9E9, 9E9, 9E9, 9E9, 9E9, 9E9]];
    CONST robtarget p16302:= [[1563.5501444937404, 22.9957521549356, 1008.500033578516], [0, 0, 1, 0], [0, 0, 0, 0], [9E9, 9E9, 9E9, 9E9, 9E9, 9E9]];
    CONST robtarget p16303:= [[1563.7317644275624, 22.396386933434258, 1008.500033578516], [0, 0, 1, 0], [0, 0, 0, 0], [9E9, 9E9, 9E9, 9E9, 9E9, 9E9]];
    CONST robtarget p16304:= [[1563.8499118427112, 22.0845151212539, 1008.500033578516], [0, 0, 1, 0], [0, 0, 0, 0], [9E9, 9E9, 9E9, 9E9, 9E9, 9E9]];
    CONST robtarget p16305:= [[1564.0375401164447, 21.4639327394908, 1008.500033578516], [0, 0, 1, 0], [0, 0, 0, 0], [9E9, 9E9, 9E9, 9E9, 9E9, 9E9]];
    CONST robtarget p16306:= [[1564.2626453473324, 20.757010672836984, 1008.500033578516], [0, 0, 1, 0], [0, 0, 0, 0], [9E9, 9E9, 9E9, 9E9, 9E9, 9E9]];
    CONST robtarget p16307:= [[1564.4266021184112, 20.35471903860835, 1008.500033578516], [0, 0, 1, 0], [0, 0, 0, 0], [9E9, 9E9, 9E9, 9E9, 9E9, 9E9]];
    CONST robtarget p16308:= [[1564.6346568991287, 19.809251624306867, 1008.500033578516], [0, 0, 1, 0], [0, 0, 0, 0], [9E9, 9E9, 9E9, 9E9, 9E9, 9E9]];
    CONST robtarget p16309:= [[1564.7613555861203, 19.408463601063943, 1008.500033578516], [0, 0, 1, 0], [0, 0, 0, 0], [9E9, 9E9, 9E9, 9E9, 9E9, 9E9]];
    CONST robtarget p16310:= [[1564.7875507803442, 19.32862098206276, 1008.500033578516], [0, 0, 1, 0], [0, 0, 0, 0], [9E9, 9E9, 9E9, 9E9, 9E9, 9E9]];
    CONST robtarget p16311:= [[1564.9419240602283, 18.679689134549832, 1008.500033578516], [0, 0, 1, 0], [0, 0, 0, 0], [9E9, 9E9, 9E9, 9E9, 9E9, 9E9]];
    CONST robtarget p16312:= [[1565.1073585052393, 17.95832784462725, 1008.500033578516], [0, 0, 1, 0], [0, 0, 0, 0], [9E9, 9E9, 9E9, 9E9, 9E9, 9E9]];
    CONST robtarget p16313:= [[1565.2748236381756, 17.390065587001274, 1008.500033578516], [0, 0, 1, 0], [0, 0, 0, 0], [9E9, 9E9, 9E9, 9E9, 9E9, 9E9]];
    CONST robtarget p16314:= [[1565.3498996361886, 17.140979099309035, 1008.500033578516], [0, 0, 1, 0], [0, 0, 0, 0], [9E9, 9E9, 9E9, 9E9, 9E9, 9E9]];
    CONST robtarget p16315:= [[1565.5335227998796, 16.404374371744325, 1008.500033578516], [0, 0, 1, 0], [0, 0, 0, 0], [9E9, 9E9, 9E9, 9E9, 9E9, 9E9]];
    CONST robtarget p16316:= [[1565.624195506827, 15.961173371755038, 1008.500033578516], [0, 0, 1, 0], [0, 0, 0, 0], [9E9, 9E9, 9E9, 9E9, 9E9, 9E9]];
    CONST robtarget p16317:= [[1565.8673733457101, 15.14454852721559, 1008.500033578516], [0, 0, 1, 0], [0, 0, 0, 0], [9E9, 9E9, 9E9, 9E9, 9E9, 9E9]];
    CONST robtarget p16318:= [[1566.0107609124025, 14.58524026253697, 1008.500033578516], [0, 0, 1, 0], [0, 0, 0, 0], [9E9, 9E9, 9E9, 9E9, 9E9, 9E9]];
    CONST robtarget p16319:= [[1566.0683622378256, 14.314339892629249, 1008.500033578516], [0, 0, 1, 0], [0, 0, 0, 0], [9E9, 9E9, 9E9, 9E9, 9E9, 9E9]];
    CONST robtarget p16320:= [[1566.2112843533641, 13.539263620215806, 1008.500033578516], [0, 0, 1, 0], [0, 0, 0, 0], [9E9, 9E9, 9E9, 9E9, 9E9, 9E9]];
    CONST robtarget p16321:= [[1566.3086465827419, 13.00486713834168, 1008.500033578516], [0, 0, 1, 0], [0, 0, 0, 0], [9E9, 9E9, 9E9, 9E9, 9E9, 9E9]];
    CONST robtarget p16322:= [[1566.3476691924363, 12.552781285095492, 1008.500033578516], [0, 0, 1, 0], [0, 0, 0, 0], [9E9, 9E9, 9E9, 9E9, 9E9, 9E9]];
    CONST robtarget p16323:= [[1566.4573876091147, 11.906837238978966, 1008.500033578516], [0, 0, 1, 0], [0, 0, 0, 0], [9E9, 9E9, 9E9, 9E9, 9E9, 9E9]];
    CONST robtarget p16324:= [[1566.557016761668, 11.480667524980774, 1008.500033578516], [0, 0, 1, 0], [0, 0, 0, 0], [9E9, 9E9, 9E9, 9E9, 9E9, 9E9]];
    CONST robtarget p16325:= [[1566.6925848685562, 10.788537359985028, 1008.500033578516], [0, 0, 1, 0], [0, 0, 0, 0], [9E9, 9E9, 9E9, 9E9, 9E9, 9E9]];
    CONST robtarget p16326:= [[1566.7186483401733, 10.595388438757439, 1008.500033578516], [0, 0, 1, 0], [0, 0, 0, 0], [9E9, 9E9, 9E9, 9E9, 9E9, 9E9]];
    CONST robtarget p16327:= [[1566.759355843255, 10.313457043957527, 1008.500033578516], [0, 0, 1, 0], [0, 0, 0, 0], [9E9, 9E9, 9E9, 9E9, 9E9, 9E9]];
    CONST robtarget p16328:= [[1566.9028437163524, 9.694455468147297, 1008.500033578516], [0, 0, 1, 0], [0, 0, 0, 0], [9E9, 9E9, 9E9, 9E9, 9E9, 9E9]];
    CONST robtarget p16329:= [[1566.9845241192043, 8.996029781929039, 1008.500033578516], [0, 0, 1, 0], [0, 0, 0, 0], [9E9, 9E9, 9E9, 9E9, 9E9, 9E9]];
    CONST robtarget p16330:= [[1567.0257565051322, 8.655019314181189, 1008.500033578516], [0, 0, 1, 0], [0, 0, 0, 0], [9E9, 9E9, 9E9, 9E9, 9E9, 9E9]];
    CONST robtarget p16331:= [[1567.0888450980012, 7.77473966150329, 1008.500033578516], [0, 0, 1, 0], [0, 0, 0, 0], [9E9, 9E9, 9E9, 9E9, 9E9, 9E9]];
    CONST robtarget p16332:= [[1567.0961196359451, 7.724676471113639, 1008.500033578516], [0, 0, 1, 0], [0, 0, 0, 0], [9E9, 9E9, 9E9, 9E9, 9E9, 9E9]];
    CONST robtarget p16333:= [[1567.1263573223182, 7.34782048852891, 1008.500033578516], [0, 0, 1, 0], [0, 0, 0, 0], [9E9, 9E9, 9E9, 9E9, 9E9, 9E9]];
    CONST robtarget p16334:= [[1567.187182522538, 6.930827962831799, 1008.500033578516], [0, 0, 1, 0], [0, 0, 0, 0], [9E9, 9E9, 9E9, 9E9, 9E9, 9E9]];
    CONST robtarget p16335:= [[1567.2608558139798, 6.38173399974815, 1008.500033578516], [0, 0, 1, 0], [0, 0, 0, 0], [9E9, 9E9, 9E9, 9E9, 9E9, 9E9]];
    CONST robtarget p16336:= [[1567.311859209369, 5.8257911094873975, 1008.500033578516], [0, 0, 1, 0], [0, 0, 0, 0], [9E9, 9E9, 9E9, 9E9, 9E9, 9E9]];
    CONST robtarget p16337:= [[1567.3927697784102, 5.2187263949316645, 1008.500033578516], [0, 0, 1, 0], [0, 0, 0, 0], [9E9, 9E9, 9E9, 9E9, 9E9, 9E9]];
    CONST robtarget p16338:= [[1567.404928013037, 5.049665351504828, 1008.500033578516], [0, 0, 1, 0], [0, 0, 0, 0], [9E9, 9E9, 9E9, 9E9, 9E9, 9E9]];
    CONST robtarget p16339:= [[1567.4183451460028, 4.883435823632425, 1008.500033578516], [0, 0, 1, 0], [0, 0, 0, 0], [9E9, 9E9, 9E9, 9E9, 9E9, 9E9]];
    CONST robtarget p16340:= [[1567.4150845750955, 4.719267795060858, 1008.500033578516], [0, 0, 1, 0], [0, 0, 0, 0], [9E9, 9E9, 9E9, 9E9, 9E9, 9E9]];
    CONST robtarget p16341:= [[1567.4208062777234, 4.273571873751578, 1008.500033578516], [0, 0, 1, 0], [0, 0, 0, 0], [9E9, 9E9, 9E9, 9E9, 9E9, 9E9]];
    CONST robtarget p16342:= [[1567.4757654489028, 3.4811400541096447, 1008.500033578516], [0, 0, 1, 0], [0, 0, 0, 0], [9E9, 9E9, 9E9, 9E9, 9E9, 9E9]];
    CONST robtarget p16343:= [[1567.4367056294195, 2.9477069778262717, 1008.500033578516], [0, 0, 1, 0], [0, 0, 0, 0], [9E9, 9E9, 9E9, 9E9, 9E9, 9E9]];
    CONST robtarget p16344:= [[1567.5457194914684, 1.656387190757144, 1008.500033578516], [0, 0, 1, 0], [0, 0, 0, 0], [9E9, 9E9, 9E9, 9E9, 9E9, 9E9]];
    CONST robtarget p16345:= [[1567.602936357975, 0.17107368758937014, 1008.500033578516], [0, 0, 1, 0], [0, 0, 0, 0], [9E9, 9E9, 9E9, 9E9, 9E9, 9E9]];
    CONST robtarget p16346:= [[1567.5996252000243, -0.2333464988671352, 1008.500033578516], [0, 0, 1, 0], [0, 0, 0, 0], [9E9, 9E9, 9E9, 9E9, 9E9, 9E9]];
    CONST robtarget p16347:= [[1567.5764487205176, -1.0042716013399087, 1008.500033578516], [0, 0, 1, 0], [0, 0, 0, 0], [9E9, 9E9, 9E9, 9E9, 9E9, 9E9]];
    CONST robtarget p16348:= [[1567.5443038388287, -1.7131925054288075, 1008.500033578516], [0, 0, 1, 0], [0, 0, 0, 0], [9E9, 9E9, 9E9, 9E9, 9E9, 9E9]];
    CONST robtarget p16349:= [[1567.527225076885, -2.2907571172341648, 1008.500033578516], [0, 0, 1, 0], [0, 0, 0, 0], [9E9, 9E9, 9E9, 9E9, 9E9, 9E9]];
    CONST robtarget p16350:= [[1567.5215536377261, -2.5821975216732653, 1008.500033578516], [0, 0, 1, 0], [0, 0, 0, 0], [9E9, 9E9, 9E9, 9E9, 9E9, 9E9]];
    CONST robtarget p16351:= [[1567.4770298997282, -2.914228557076143, 1008.500033578516], [0, 0, 1, 0], [0, 0, 0, 0], [9E9, 9E9, 9E9, 9E9, 9E9, 9E9]];
    CONST robtarget p16352:= [[1567.4501830214706, -4.186518220217167, 1008.500033578516], [0, 0, 1, 0], [0, 0, 0, 0], [9E9, 9E9, 9E9, 9E9, 9E9, 9E9]];
    CONST robtarget p16353:= [[1567.4500918483013, -4.212558993292518, 1008.500033578516], [0, 0, 1, 0], [0, 0, 0, 0], [9E9, 9E9, 9E9, 9E9, 9E9, 9E9]];
    CONST robtarget p16354:= [[1567.4182280014718, -5.03184153844596, 1008.500033578516], [0, 0, 1, 0], [0, 0, 0, 0], [9E9, 9E9, 9E9, 9E9, 9E9, 9E9]];
    CONST robtarget p16355:= [[1567.3218972371537, -5.966021411702187, 1008.500033578516], [0, 0, 1, 0], [0, 0, 0, 0], [9E9, 9E9, 9E9, 9E9, 9E9, 9E9]];
    CONST robtarget p16356:= [[1567.2156476842401, -6.786579513796731, 1008.500033578516], [0, 0, 1, 0], [0, 0, 0, 0], [9E9, 9E9, 9E9, 9E9, 9E9, 9E9]];
    CONST robtarget p16357:= [[1567.2141720488098, -6.802453830611313, 1008.500033578516], [0, 0, 1, 0], [0, 0, 0, 0], [9E9, 9E9, 9E9, 9E9, 9E9, 9E9]];
    CONST robtarget p16358:= [[1567.1661698693526, -7.2916271019348855, 1008.500033578516], [0, 0, 1, 0], [0, 0, 0, 0], [9E9, 9E9, 9E9, 9E9, 9E9, 9E9]];
    CONST robtarget p16359:= [[1567.107078491758, -7.906428738627852, 1008.500033578516], [0, 0, 1, 0], [0, 0, 0, 0], [9E9, 9E9, 9E9, 9E9, 9E9, 9E9]];
    CONST robtarget p16360:= [[1567.0976389272619, -7.970196105973528, 1008.500033578516], [0, 0, 1, 0], [0, 0, 0, 0], [9E9, 9E9, 9E9, 9E9, 9E9, 9E9]];
    CONST robtarget p16361:= [[1567.0763958214857, -8.13452460629152, 1008.500033578516], [0, 0, 1, 0], [0, 0, 0, 0], [9E9, 9E9, 9E9, 9E9, 9E9, 9E9]];
    CONST robtarget p16362:= [[1567.0032710585472, -8.864633267259137, 1008.500033578516], [0, 0, 1, 0], [0, 0, 0, 0], [9E9, 9E9, 9E9, 9E9, 9E9, 9E9]];
    CONST robtarget p16363:= [[1566.858153752501, -9.569953991234712, 1008.500033578516], [0, 0, 1, 0], [0, 0, 0, 0], [9E9, 9E9, 9E9, 9E9, 9E9, 9E9]];
    CONST robtarget p16364:= [[1566.822304017215, -9.88902746248278, 1008.500033578516], [0, 0, 1, 0], [0, 0, 0, 0], [9E9, 9E9, 9E9, 9E9, 9E9, 9E9]];
    CONST robtarget p16365:= [[1566.7434027263198, -10.380313773471435, 1008.500033578516], [0, 0, 1, 0], [0, 0, 0, 0], [9E9, 9E9, 9E9, 9E9, 9E9, 9E9]];
    CONST robtarget p16366:= [[1566.7350925866974, -10.434402872814687, 1008.500033578516], [0, 0, 1, 0], [0, 0, 0, 0], [9E9, 9E9, 9E9, 9E9, 9E9, 9E9]];
    CONST robtarget p16367:= [[1566.7001887648921, -10.584355998866883, 1008.500033578516], [0, 0, 1, 0], [0, 0, 0, 0], [9E9, 9E9, 9E9, 9E9, 9E9, 9E9]];
    CONST robtarget p16368:= [[1566.5610591434183, -11.470137452439609, 1008.500033578516], [0, 0, 1, 0], [0, 0, 0, 0], [9E9, 9E9, 9E9, 9E9, 9E9, 9E9]];
    CONST robtarget p16369:= [[1566.5224846565243, -11.764955218516903, 1008.500033578516], [0, 0, 1, 0], [0, 0, 0, 0], [9E9, 9E9, 9E9, 9E9, 9E9, 9E9]];
    CONST robtarget p16370:= [[1566.5045611147373, -11.941697210548547, 1008.500033578516], [0, 0, 1, 0], [0, 0, 0, 0], [9E9, 9E9, 9E9, 9E9, 9E9, 9E9]];
    CONST robtarget p16371:= [[1566.4581977985677, -12.17188055628673, 1008.500033578516], [0, 0, 1, 0], [0, 0, 0, 0], [9E9, 9E9, 9E9, 9E9, 9E9, 9E9]];
    CONST robtarget p16372:= [[1566.3267161120975, -12.69298893434528, 1008.500033578516], [0, 0, 1, 0], [0, 0, 0, 0], [9E9, 9E9, 9E9, 9E9, 9E9, 9E9]];
    CONST robtarget p16373:= [[1566.1963110650354, -13.621644659694624, 1008.500033578516], [0, 0, 1, 0], [0, 0, 0, 0], [9E9, 9E9, 9E9, 9E9, 9E9, 9E9]];
    CONST robtarget p16374:= [[1566.0032788922804, -14.329814399815355, 1008.500033578516], [0, 0, 1, 0], [0, 0, 0, 0], [9E9, 9E9, 9E9, 9E9, 9E9, 9E9]];
    CONST robtarget p16375:= [[1565.8277890147153, -15.306455398062567, 1008.500033578516], [0, 0, 1, 0], [0, 0, 0, 0], [9E9, 9E9, 9E9, 9E9, 9E9, 9E9]];
    CONST robtarget p16376:= [[1565.7307064274744, -15.629971482187045, 1008.500033578516], [0, 0, 1, 0], [0, 0, 0, 0], [9E9, 9E9, 9E9, 9E9, 9E9, 9E9]];
    CONST robtarget p16377:= [[1565.5803798315765, -16.29030575129898, 1008.500033578516], [0, 0, 1, 0], [0, 0, 0, 0], [9E9, 9E9, 9E9, 9E9, 9E9, 9E9]];
    CONST robtarget p16378:= [[1565.4348993989101, -16.825881959955282, 1008.500033578516], [0, 0, 1, 0], [0, 0, 0, 0], [9E9, 9E9, 9E9, 9E9, 9E9, 9E9]];
    CONST robtarget p16379:= [[1565.4122134439583, -16.910171452684693, 1008.500033578516], [0, 0, 1, 0], [0, 0, 0, 0], [9E9, 9E9, 9E9, 9E9, 9E9, 9E9]];
    CONST robtarget p16380:= [[1565.266377187281, -17.403969020238172, 1008.500033578516], [0, 0, 1, 0], [0, 0, 0, 0], [9E9, 9E9, 9E9, 9E9, 9E9, 9E9]];
    CONST robtarget p16381:= [[1565.1208792614082, -18.050586130127762, 1008.500033578516], [0, 0, 1, 0], [0, 0, 0, 0], [9E9, 9E9, 9E9, 9E9, 9E9, 9E9]];
    CONST robtarget p16382:= [[1564.928290599989, -18.791194179873244, 1008.500033578516], [0, 0, 1, 0], [0, 0, 0, 0], [9E9, 9E9, 9E9, 9E9, 9E9, 9E9]];
    CONST robtarget p16383:= [[1564.7922394833663, -19.17392557074421, 1008.500033578516], [0, 0, 1, 0], [0, 0, 0, 0], [9E9, 9E9, 9E9, 9E9, 9E9, 9E9]];
    CONST robtarget p16384:= [[1564.6528259746033, -19.693394650432147, 1008.500033578516], [0, 0, 1, 0], [0, 0, 0, 0], [9E9, 9E9, 9E9, 9E9, 9E9, 9E9]];
    CONST robtarget p16385:= [[1564.5398375326952, -20.0516761286246, 1008.500033578516], [0, 0, 1, 0], [0, 0, 0, 0], [9E9, 9E9, 9E9, 9E9, 9E9, 9E9]];
    CONST robtarget p16386:= [[1564.4918016132115, -20.16753515783025, 1008.500033578516], [0, 0, 1, 0], [0, 0, 0, 0], [9E9, 9E9, 9E9, 9E9, 9E9, 9E9]];
    CONST robtarget p16387:= [[1564.2565822724112, -20.871056841580696, 1008.500033578516], [0, 0, 1, 0], [0, 0, 0, 0], [9E9, 9E9, 9E9, 9E9, 9E9, 9E9]];
    CONST robtarget p16388:= [[1564.2158164705, -21.04280335201566, 1008.500033578516], [0, 0, 1, 0], [0, 0, 0, 0], [9E9, 9E9, 9E9, 9E9, 9E9, 9E9]];
    CONST robtarget p16389:= [[1564.0647728470262, -21.46671406410166, 1008.500033578516], [0, 0, 1, 0], [0, 0, 0, 0], [9E9, 9E9, 9E9, 9E9, 9E9, 9E9]];
    CONST robtarget p16390:= [[1563.8142774391404, -22.15568406909103, 1008.500033578516], [0, 0, 1, 0], [0, 0, 0, 0], [9E9, 9E9, 9E9, 9E9, 9E9, 9E9]];
    CONST robtarget p16391:= [[1563.492756089425, -23.12268003116379, 1008.500033578516], [0, 0, 1, 0], [0, 0, 0, 0], [9E9, 9E9, 9E9, 9E9, 9E9, 9E9]];
    CONST robtarget p16392:= [[1563.311190603778, -23.653669559703495, 1008.500033578516], [0, 0, 1, 0], [0, 0, 0, 0], [9E9, 9E9, 9E9, 9E9, 9E9, 9E9]];
    CONST robtarget p16393:= [[1563.1204488123317, -24.1253488909783, 1008.500033578516], [0, 0, 1, 0], [0, 0, 0, 0], [9E9, 9E9, 9E9, 9E9, 9E9, 9E9]];
    CONST robtarget p16394:= [[1562.956092777694, -24.58260761287665, 1008.500033578516], [0, 0, 1, 0], [0, 0, 0, 0], [9E9, 9E9, 9E9, 9E9, 9E9, 9E9]];
    CONST robtarget p16395:= [[1562.8290753792662, -24.897857668625427, 1008.500033578516], [0, 0, 1, 0], [0, 0, 0, 0], [9E9, 9E9, 9E9, 9E9, 9E9, 9E9]];
    CONST robtarget p16396:= [[1562.3614724756612, -26.01944537119558, 1008.500033578516], [0, 0, 1, 0], [0, 0, 0, 0], [9E9, 9E9, 9E9, 9E9, 9E9, 9E9]];
    CONST robtarget p16397:= [[1562.1937679544649, -26.408007145605254, 1008.500033578516], [0, 0, 1, 0], [0, 0, 0, 0], [9E9, 9E9, 9E9, 9E9, 9E9, 9E9]];
    CONST robtarget p16398:= [[1561.7538610476063, -27.428629634373742, 1008.500033578516], [0, 0, 1, 0], [0, 0, 0, 0], [9E9, 9E9, 9E9, 9E9, 9E9, 9E9]];
    CONST robtarget p16399:= [[1561.5574779491817, -27.862286240525528, 1008.500033578516], [0, 0, 1, 0], [0, 0, 0, 0], [9E9, 9E9, 9E9, 9E9, 9E9, 9E9]];
    CONST robtarget p16400:= [[1561.4799670574819, -28.021933888720568, 1008.500033578516], [0, 0, 1, 0], [0, 0, 0, 0], [9E9, 9E9, 9E9, 9E9, 9E9, 9E9]];
    CONST robtarget p16401:= [[1561.2417653428213, -28.625868436615754, 1008.500033578516], [0, 0, 1, 0], [0, 0, 0, 0], [9E9, 9E9, 9E9, 9E9, 9E9, 9E9]];
    CONST robtarget p16402:= [[1561.1374870704649, -28.838547515831678, 1008.500033578516], [0, 0, 1, 0], [0, 0, 0, 0], [9E9, 9E9, 9E9, 9E9, 9E9, 9E9]];
    CONST robtarget p16403:= [[1560.9491800643614, -29.218947012338788, 1008.500033578516], [0, 0, 1, 0], [0, 0, 0, 0], [9E9, 9E9, 9E9, 9E9, 9E9, 9E9]];
    CONST robtarget p16404:= [[1560.5405023196652, -30.01764042738396, 1008.500033578516], [0, 0, 1, 0], [0, 0, 0, 0], [9E9, 9E9, 9E9, 9E9, 9E9, 9E9]];
    CONST robtarget p16405:= [[1559.9668823667403, -31.110955980969457, 1008.500033578516], [0, 0, 1, 0], [0, 0, 0, 0], [9E9, 9E9, 9E9, 9E9, 9E9, 9E9]];
    CONST robtarget p16406:= [[1559.7614657530528, -31.51521018069753, 1008.500033578516], [0, 0, 1, 0], [0, 0, 0, 0], [9E9, 9E9, 9E9, 9E9, 9E9, 9E9]];
    CONST robtarget p16407:= [[1559.6765787856314, -31.65441340476356, 1008.500033578516], [0, 0, 1, 0], [0, 0, 0, 0], [9E9, 9E9, 9E9, 9E9, 9E9, 9E9]];
    CONST robtarget p16408:= [[1559.1729065895179, -32.687470690677124, 1008.500033578516], [0, 0, 1, 0], [0, 0, 0, 0], [9E9, 9E9, 9E9, 9E9, 9E9, 9E9]];
    CONST robtarget p16409:= [[1558.8248061573734, -33.272769205948926, 1008.500033578516], [0, 0, 1, 0], [0, 0, 0, 0], [9E9, 9E9, 9E9, 9E9, 9E9, 9E9]];
    CONST robtarget p16410:= [[1558.7170316785964, -33.48350727630887, 1008.500033578516], [0, 0, 1, 0], [0, 0, 0, 0], [9E9, 9E9, 9E9, 9E9, 9E9, 9E9]];
    CONST robtarget p16411:= [[1558.5283776227645, -33.8005388724041, 1008.500033578516], [0, 0, 1, 0], [0, 0, 0, 0], [9E9, 9E9, 9E9, 9E9, 9E9, 9E9]];
    CONST robtarget p16412:= [[1557.9007907694538, -34.79474767324494, 1008.500033578516], [0, 0, 1, 0], [0, 0, 0, 0], [9E9, 9E9, 9E9, 9E9, 9E9, 9E9]];
    CONST robtarget p16413:= [[1557.734715904432, -35.06997527692259, 1008.500033578516], [0, 0, 1, 0], [0, 0, 0, 0], [9E9, 9E9, 9E9, 9E9, 9E9, 9E9]];
    CONST robtarget p16414:= [[1557.1278930218937, -35.99515743573169, 1008.500033578516], [0, 0, 1, 0], [0, 0, 0, 0], [9E9, 9E9, 9E9, 9E9, 9E9, 9E9]];
    CONST robtarget p16415:= [[1556.8449238374697, -36.56850518632186, 1008.500033578516], [0, 0, 1, 0], [0, 0, 0, 0], [9E9, 9E9, 9E9, 9E9, 9E9, 9E9]];
    CONST robtarget p16416:= [[1556.6192334752711, -36.9376058061577, 1008.500033578516], [0, 0, 1, 0], [0, 0, 0, 0], [9E9, 9E9, 9E9, 9E9, 9E9, 9E9]];
    CONST robtarget p16417:= [[1556.1854365806462, -37.526816919343766, 1008.500033578516], [0, 0, 1, 0], [0, 0, 0, 0], [9E9, 9E9, 9E9, 9E9, 9E9, 9E9]];
    CONST robtarget p16418:= [[1555.9664458434193, -37.84222699391139, 1008.500033578516], [0, 0, 1, 0], [0, 0, 0, 0], [9E9, 9E9, 9E9, 9E9, 9E9, 9E9]];
    CONST robtarget p16419:= [[1555.743215660483, -38.21750364385949, 1008.500033578516], [0, 0, 1, 0], [0, 0, 0, 0], [9E9, 9E9, 9E9, 9E9, 9E9, 9E9]];
    CONST robtarget p16420:= [[1555.5605751513008, -38.46469865336096, 1008.500033578516], [0, 0, 1, 0], [0, 0, 0, 0], [9E9, 9E9, 9E9, 9E9, 9E9, 9E9]];
    CONST robtarget p16421:= [[1555.2652518245145, -38.88488415285963, 1008.500033578516], [0, 0, 1, 0], [0, 0, 0, 0], [9E9, 9E9, 9E9, 9E9, 9E9, 9E9]];
    CONST robtarget p16422:= [[1554.960735477367, -39.229439935219645, 1008.500033578516], [0, 0, 1, 0], [0, 0, 0, 0], [9E9, 9E9, 9E9, 9E9, 9E9, 9E9]];
    CONST robtarget p16423:= [[1554.2685702291799, -40.2681929540489, 1008.500033578516], [0, 0, 1, 0], [0, 0, 0, 0], [9E9, 9E9, 9E9, 9E9, 9E9, 9E9]];
    CONST robtarget p16424:= [[1553.5804835921567, -41.220486388103936, 1008.500033578516], [0, 0, 1, 0], [0, 0, 0, 0], [9E9, 9E9, 9E9, 9E9, 9E9, 9E9]];
    CONST robtarget p16425:= [[1552.9648806741725, -41.975329128526134, 1008.500033578516], [0, 0, 1, 0], [0, 0, 0, 0], [9E9, 9E9, 9E9, 9E9, 9E9, 9E9]];
    CONST robtarget p16426:= [[1552.6148404874268, -42.41293677600321, 1008.500033578516], [0, 0, 1, 0], [0, 0, 0, 0], [9E9, 9E9, 9E9, 9E9, 9E9, 9E9]];
    CONST robtarget p16427:= [[1552.4070155145264, -42.63878690068773, 1008.500033578516], [0, 0, 1, 0], [0, 0, 0, 0], [9E9, 9E9, 9E9, 9E9, 9E9, 9E9]];
    CONST robtarget p16428:= [[1552.258172215424, -42.81701581665671, 1008.500033578516], [0, 0, 1, 0], [0, 0, 0, 0], [9E9, 9E9, 9E9, 9E9, 9E9, 9E9]];
    CONST robtarget p16429:= [[1551.923499091037, -43.24052564096954, 1008.500033578516], [0, 0, 1, 0], [0, 0, 0, 0], [9E9, 9E9, 9E9, 9E9, 9E9, 9E9]];
    CONST robtarget p16430:= [[1551.8513608885175, -43.32487640285498, 1008.500033578516], [0, 0, 1, 0], [0, 0, 0, 0], [9E9, 9E9, 9E9, 9E9, 9E9, 9E9]];
    CONST robtarget p16431:= [[1551.6004728821138, -43.616104039139046, 1008.500033578516], [0, 0, 1, 0], [0, 0, 0, 0], [9E9, 9E9, 9E9, 9E9, 9E9, 9E9]];
    CONST robtarget p16432:= [[1551.157756769762, -44.13840851529652, 1008.500033578516], [0, 0, 1, 0], [0, 0, 0, 0], [9E9, 9E9, 9E9, 9E9, 9E9, 9E9]];
    CONST robtarget p16433:= [[1550.6833501804322, -44.68963522751863, 1008.500033578516], [0, 0, 1, 0], [0, 0, 0, 0], [9E9, 9E9, 9E9, 9E9, 9E9, 9E9]];
    CONST robtarget p16434:= [[1550.3880441243628, -45.07551085563114, 1008.500033578516], [0, 0, 1, 0], [0, 0, 0, 0], [9E9, 9E9, 9E9, 9E9, 9E9, 9E9]];
    CONST robtarget p16435:= [[1549.924854559153, -45.55032063903374, 1008.500033578516], [0, 0, 1, 0], [0, 0, 0, 0], [9E9, 9E9, 9E9, 9E9, 9E9, 9E9]];
    CONST robtarget p16436:= [[1549.6005328863569, -45.90741343238179, 1008.500033578516], [0, 0, 1, 0], [0, 0, 0, 0], [9E9, 9E9, 9E9, 9E9, 9E9, 9E9]];
    CONST robtarget p16437:= [[1549.0384525871661, -46.47116908743163, 1008.500033578516], [0, 0, 1, 0], [0, 0, 0, 0], [9E9, 9E9, 9E9, 9E9, 9E9, 9E9]];
    CONST robtarget p16438:= [[1548.9457915056446, -46.571228056661624, 1008.500033578516], [0, 0, 1, 0], [0, 0, 0, 0], [9E9, 9E9, 9E9, 9E9, 9E9, 9E9]];
    CONST robtarget p16439:= [[1548.3292327208048, -47.1930047574031, 1008.500033578516], [0, 0, 1, 0], [0, 0, 0, 0], [9E9, 9E9, 9E9, 9E9, 9E9, 9E9]];
    CONST robtarget p16440:= [[1548.1595309261475, -47.383495891184126, 1008.500033578516], [0, 0, 1, 0], [0, 0, 0, 0], [9E9, 9E9, 9E9, 9E9, 9E9, 9E9]];
    CONST robtarget p16441:= [[1547.7379579972187, -47.81826169916996, 1008.500033578516], [0, 0, 1, 0], [0, 0, 0, 0], [9E9, 9E9, 9E9, 9E9, 9E9, 9E9]];
    CONST robtarget p16442:= [[1547.1958239233604, -48.39615411886057, 1008.500033578516], [0, 0, 1, 0], [0, 0, 0, 0], [9E9, 9E9, 9E9, 9E9, 9E9, 9E9]];
    CONST robtarget p16443:= [[1546.9143330553438, -48.679593953919905, 1008.500033578516], [0, 0, 1, 0], [0, 0, 0, 0], [9E9, 9E9, 9E9, 9E9, 9E9, 9E9]];
    CONST robtarget p16444:= [[1546.6443913989078, -48.905652635398226, 1008.500033578516], [0, 0, 1, 0], [0, 0, 0, 0], [9E9, 9E9, 9E9, 9E9, 9E9, 9E9]];
    CONST robtarget p16445:= [[1546.1729667960387, -49.35389603808956, 1008.500033578516], [0, 0, 1, 0], [0, 0, 0, 0], [9E9, 9E9, 9E9, 9E9, 9E9, 9E9]];
    CONST robtarget p16446:= [[1546.035262349947, -49.46309983989453, 1008.500033578516], [0, 0, 1, 0], [0, 0, 0, 0], [9E9, 9E9, 9E9, 9E9, 9E9, 9E9]];
    CONST robtarget p16447:= [[1545.5052034574992, -49.94193148421713, 1008.500033578516], [0, 0, 1, 0], [0, 0, 0, 0], [9E9, 9E9, 9E9, 9E9, 9E9, 9E9]];
    CONST robtarget p16448:= [[1545.3151913922222, -50.08617153750216, 1008.500033578516], [0, 0, 1, 0], [0, 0, 0, 0], [9E9, 9E9, 9E9, 9E9, 9E9, 9E9]];
    CONST robtarget p16449:= [[1544.666470799138, -50.686922215694096, 1008.500033578516], [0, 0, 1, 0], [0, 0, 0, 0], [9E9, 9E9, 9E9, 9E9, 9E9, 9E9]];
    CONST robtarget p16450:= [[1544.4925268504933, -50.832028773913336, 1008.500033578516], [0, 0, 1, 0], [0, 0, 0, 0], [9E9, 9E9, 9E9, 9E9, 9E9, 9E9]];
    CONST robtarget p16451:= [[1543.835047131417, -51.45475774648632, 1008.500033578516], [0, 0, 1, 0], [0, 0, 0, 0], [9E9, 9E9, 9E9, 9E9, 9E9, 9E9]];
    CONST robtarget p16452:= [[1543.232872353631, -51.979068464882985, 1008.500033578516], [0, 0, 1, 0], [0, 0, 0, 0], [9E9, 9E9, 9E9, 9E9, 9E9, 9E9]];
    CONST robtarget p16453:= [[1542.979265905555, -52.14852814309041, 1008.500033578516], [0, 0, 1, 0], [0, 0, 0, 0], [9E9, 9E9, 9E9, 9E9, 9E9, 9E9]];
    CONST robtarget p16454:= [[1542.3619394588115, -52.61447291408469, 1008.500033578516], [0, 0, 1, 0], [0, 0, 0, 0], [9E9, 9E9, 9E9, 9E9, 9E9, 9E9]];
    CONST robtarget p16455:= [[1542.2460152583233, -52.703197999201805, 1008.500033578516], [0, 0, 1, 0], [0, 0, 0, 0], [9E9, 9E9, 9E9, 9E9, 9E9, 9E9]];
    CONST robtarget p16456:= [[1541.5332956120515, -53.25616091096338, 1008.500033578516], [0, 0, 1, 0], [0, 0, 0, 0], [9E9, 9E9, 9E9, 9E9, 9E9, 9E9]];
    CONST robtarget p16457:= [[1541.146287510733, -53.589127073170694, 1008.500033578516], [0, 0, 1, 0], [0, 0, 0, 0], [9E9, 9E9, 9E9, 9E9, 9E9, 9E9]];
    CONST robtarget p16458:= [[1541.081604301113, -53.633756733544715, 1008.500033578516], [0, 0, 1, 0], [0, 0, 0, 0], [9E9, 9E9, 9E9, 9E9, 9E9, 9E9]];
    CONST robtarget p16459:= [[1540.4802364821335, -54.08844227126839, 1008.500033578516], [0, 0, 1, 0], [0, 0, 0, 0], [9E9, 9E9, 9E9, 9E9, 9E9, 9E9]];
    CONST robtarget p16460:= [[1540.1800374233007, -54.321997607572015, 1008.500033578516], [0, 0, 1, 0], [0, 0, 0, 0], [9E9, 9E9, 9E9, 9E9, 9E9, 9E9]];
    CONST robtarget p16461:= [[1539.6359252511663, -54.75999173971934, 1008.500033578516], [0, 0, 1, 0], [0, 0, 0, 0], [9E9, 9E9, 9E9, 9E9, 9E9, 9E9]];
    CONST robtarget p16462:= [[1539.2306352546473, -55.05579398383851, 1008.500033578516], [0, 0, 1, 0], [0, 0, 0, 0], [9E9, 9E9, 9E9, 9E9, 9E9, 9E9]];
    CONST robtarget p16463:= [[1539.0092497000037, -55.194430091586426, 1008.500033578516], [0, 0, 1, 0], [0, 0, 0, 0], [9E9, 9E9, 9E9, 9E9, 9E9, 9E9]];
    CONST robtarget p16464:= [[1538.6291054513208, -55.43239565248703, 1008.500033578516], [0, 0, 1, 0], [0, 0, 0, 0], [9E9, 9E9, 9E9, 9E9, 9E9, 9E9]];
    CONST robtarget p16465:= [[1537.9549290658374, -55.9088924917568, 1008.500033578516], [0, 0, 1, 0], [0, 0, 0, 0], [9E9, 9E9, 9E9, 9E9, 9E9, 9E9]];
    CONST robtarget p16466:= [[1537.4199907475006, -56.231207550169636, 1008.500033578516], [0, 0, 1, 0], [0, 0, 0, 0], [9E9, 9E9, 9E9, 9E9, 9E9, 9E9]];
    CONST robtarget p16467:= [[1536.8993486956372, -56.610936238859146, 1008.500033578516], [0, 0, 1, 0], [0, 0, 0, 0], [9E9, 9E9, 9E9, 9E9, 9E9, 9E9]];
    CONST robtarget p16468:= [[1536.4733124351685, -56.87723698342805, 1008.500033578516], [0, 0, 1, 0], [0, 0, 0, 0], [9E9, 9E9, 9E9, 9E9, 9E9, 9E9]];
    CONST robtarget p16469:= [[1535.9984237331305, -57.20669409955457, 1008.500033578516], [0, 0, 1, 0], [0, 0, 0, 0], [9E9, 9E9, 9E9, 9E9, 9E9, 9E9]];
    CONST robtarget p16470:= [[1535.1073962123558, -57.761733743279194, 1008.500033578516], [0, 0, 1, 0], [0, 0, 0, 0], [9E9, 9E9, 9E9, 9E9, 9E9, 9E9]];
    CONST robtarget p16471:= [[1534.8684534841962, -57.88942958975414, 1008.500033578516], [0, 0, 1, 0], [0, 0, 0, 0], [9E9, 9E9, 9E9, 9E9, 9E9, 9E9]];
    CONST robtarget p16472:= [[1534.3772605610975, -58.130636737045435, 1008.500033578516], [0, 0, 1, 0], [0, 0, 0, 0], [9E9, 9E9, 9E9, 9E9, 9E9, 9E9]];
    CONST robtarget p16473:= [[1533.836152879501, -58.47449108012872, 1008.500033578516], [0, 0, 1, 0], [0, 0, 0, 0], [9E9, 9E9, 9E9, 9E9, 9E9, 9E9]];
    CONST robtarget p16474:= [[1533.4384140498926, -58.69690751218587, 1008.500033578516], [0, 0, 1, 0], [0, 0, 0, 0], [9E9, 9E9, 9E9, 9E9, 9E9, 9E9]];
    CONST robtarget p16475:= [[1533.1468546931053, -58.882826075620684, 1008.500033578516], [0, 0, 1, 0], [0, 0, 0, 0], [9E9, 9E9, 9E9, 9E9, 9E9, 9E9]];
    CONST robtarget p16476:= [[1532.796846706207, -59.0811635467455, 1008.500033578516], [0, 0, 1, 0], [0, 0, 0, 0], [9E9, 9E9, 9E9, 9E9, 9E9, 9E9]];
    CONST robtarget p16477:= [[1532.3193767293687, -59.315608750347955, 1008.500033578516], [0, 0, 1, 0], [0, 0, 0, 0], [9E9, 9E9, 9E9, 9E9, 9E9, 9E9]];
    CONST robtarget p16478:= [[1531.9809775802764, -59.50728130055101, 1008.500033578516], [0, 0, 1, 0], [0, 0, 0, 0], [9E9, 9E9, 9E9, 9E9, 9E9, 9E9]];
    CONST robtarget p16479:= [[1531.8538063205563, -59.57735685973228, 1008.500033578516], [0, 0, 1, 0], [0, 0, 0, 0], [9E9, 9E9, 9E9, 9E9, 9E9, 9E9]];
    CONST robtarget p16480:= [[1531.2081790483692, -59.92959381362322, 1008.500033578516], [0, 0, 1, 0], [0, 0, 0, 0], [9E9, 9E9, 9E9, 9E9, 9E9, 9E9]];
    CONST robtarget p16481:= [[1530.8889468471634, -60.13104817456848, 1008.500033578516], [0, 0, 1, 0], [0, 0, 0, 0], [9E9, 9E9, 9E9, 9E9, 9E9, 9E9]];
    CONST robtarget p16482:= [[1529.9233817429597, -60.5929213076424, 1008.500033578516], [0, 0, 1, 0], [0, 0, 0, 0], [9E9, 9E9, 9E9, 9E9, 9E9, 9E9]];
    CONST robtarget p16483:= [[1529.2459335521846, -60.89534954616866, 1008.500033578516], [0, 0, 1, 0], [0, 0, 0, 0], [9E9, 9E9, 9E9, 9E9, 9E9, 9E9]];
    CONST robtarget p16484:= [[1528.7088751212204, -61.16772195339584, 1008.500033578516], [0, 0, 1, 0], [0, 0, 0, 0], [9E9, 9E9, 9E9, 9E9, 9E9, 9E9]];
    CONST robtarget p16485:= [[1528.5003394958958, -61.25513766115041, 1008.500033578516], [0, 0, 1, 0], [0, 0, 0, 0], [9E9, 9E9, 9E9, 9E9, 9E9, 9E9]];
    CONST robtarget p16486:= [[1528.050719450163, -61.47685247769042, 1008.500033578516], [0, 0, 1, 0], [0, 0, 0, 0], [9E9, 9E9, 9E9, 9E9, 9E9, 9E9]];
    CONST robtarget p16487:= [[1527.096231482812, -61.92279455652607, 1008.500033578516], [0, 0, 1, 0], [0, 0, 0, 0], [9E9, 9E9, 9E9, 9E9, 9E9, 9E9]];
    CONST robtarget p16488:= [[1526.8432896592992, -62.01901726825236, 1008.500033578516], [0, 0, 1, 0], [0, 0, 0, 0], [9E9, 9E9, 9E9, 9E9, 9E9, 9E9]];
    CONST robtarget p16489:= [[1526.1677384642423, -62.291928592178074, 1008.500033578516], [0, 0, 1, 0], [0, 0, 0, 0], [9E9, 9E9, 9E9, 9E9, 9E9, 9E9]];
    CONST robtarget p16490:= [[1525.9183750079558, -62.41826126692946, 1008.500033578516], [0, 0, 1, 0], [0, 0, 0, 0], [9E9, 9E9, 9E9, 9E9, 9E9, 9E9]];
    CONST robtarget p16491:= [[1524.7628238570912, -62.87204695974521, 1008.500033578516], [0, 0, 1, 0], [0, 0, 0, 0], [9E9, 9E9, 9E9, 9E9, 9E9, 9E9]];
    CONST robtarget p16492:= [[1524.4080277925307, -62.982154701176825, 1008.500033578516], [0, 0, 1, 0], [0, 0, 0, 0], [9E9, 9E9, 9E9, 9E9, 9E9, 9E9]];
    CONST robtarget p16493:= [[1523.7066652384433, -63.277821216605716, 1008.500033578516], [0, 0, 1, 0], [0, 0, 0, 0], [9E9, 9E9, 9E9, 9E9, 9E9, 9E9]];
    CONST robtarget p16494:= [[1523.077946184649, -63.51798103031585, 1008.500033578516], [0, 0, 1, 0], [0, 0, 0, 0], [9E9, 9E9, 9E9, 9E9, 9E9, 9E9]];
    CONST robtarget p16495:= [[1521.9556816246177, -63.942844750935045, 1008.500033578516], [0, 0, 1, 0], [0, 0, 0, 0], [9E9, 9E9, 9E9, 9E9, 9E9, 9E9]];
    CONST robtarget p16496:= [[1520.954563257394, -64.25794953131775, 1008.500033578516], [0, 0, 1, 0], [0, 0, 0, 0], [9E9, 9E9, 9E9, 9E9, 9E9, 9E9]];
    CONST robtarget p16497:= [[1520.597482798287, -64.34822457348616, 1008.500033578516], [0, 0, 1, 0], [0, 0, 0, 0], [9E9, 9E9, 9E9, 9E9, 9E9, 9E9]];
    CONST robtarget p16498:= [[1520.385536132991, -64.41077368477039, 1008.500033578516], [0, 0, 1, 0], [0, 0, 0, 0], [9E9, 9E9, 9E9, 9E9, 9E9, 9E9]];
    CONST robtarget p16499:= [[1519.8811090089785, -64.54515291203202, 1008.500033578516], [0, 0, 1, 0], [0, 0, 0, 0], [9E9, 9E9, 9E9, 9E9, 9E9, 9E9]];
    CONST robtarget p16500:= [[1519.1033258690256, -64.81836352173941, 1008.500033578516], [0, 0, 1, 0], [0, 0, 0, 0], [9E9, 9E9, 9E9, 9E9, 9E9, 9E9]];
    CONST robtarget p16501:= [[1518.8001739584358, -64.90616216584532, 1008.500033578516], [0, 0, 1, 0], [0, 0, 0, 0], [9E9, 9E9, 9E9, 9E9, 9E9, 9E9]];
    CONST robtarget p16502:= [[1518.483403147394, -65.00050395501579, 1008.500033578516], [0, 0, 1, 0], [0, 0, 0, 0], [9E9, 9E9, 9E9, 9E9, 9E9, 9E9]];
    CONST robtarget p16503:= [[1517.483089575373, -65.30024754734559, 1008.500033578516], [0, 0, 1, 0], [0, 0, 0, 0], [9E9, 9E9, 9E9, 9E9, 9E9, 9E9]];
    CONST robtarget p16504:= [[1516.872817030224, -65.459735935602, 1008.500033578516], [0, 0, 1, 0], [0, 0, 0, 0], [9E9, 9E9, 9E9, 9E9, 9E9, 9E9]];
    CONST robtarget p16505:= [[1516.4655956672862, -65.54659362808714, 1008.500033578516], [0, 0, 1, 0], [0, 0, 0, 0], [9E9, 9E9, 9E9, 9E9, 9E9, 9E9]];
    CONST robtarget p16506:= [[1516.0895359366395, -65.61955910046744, 1008.500033578516], [0, 0, 1, 0], [0, 0, 0, 0], [9E9, 9E9, 9E9, 9E9, 9E9, 9E9]];
    CONST robtarget p16507:= [[1516.0505137705593, -65.62800517390173, 1008.500033578516], [0, 0, 1, 0], [0, 0, 0, 0], [9E9, 9E9, 9E9, 9E9, 9E9, 9E9]];
    CONST robtarget p16508:= [[1515.4876219206121, -65.76610922037688, 1008.500033578516], [0, 0, 1, 0], [0, 0, 0, 0], [9E9, 9E9, 9E9, 9E9, 9E9, 9E9]];
    CONST robtarget p16509:= [[1514.2733868896114, -66.04479228917646, 1008.500033578516], [0, 0, 1, 0], [0, 0, 0, 0], [9E9, 9E9, 9E9, 9E9, 9E9, 9E9]];
    CONST robtarget p16510:= [[1514.1050063069747, -66.09062647308582, 1008.500033578516], [0, 0, 1, 0], [0, 0, 0, 0], [9E9, 9E9, 9E9, 9E9, 9E9, 9E9]];
    CONST robtarget p16511:= [[1513.416484758131, -66.22511552470365, 1008.500033578516], [0, 0, 1, 0], [0, 0, 0, 0], [9E9, 9E9, 9E9, 9E9, 9E9, 9E9]];
    CONST robtarget p16512:= [[1512.8270518503693, -66.31778803621917, 1008.500033578516], [0, 0, 1, 0], [0, 0, 0, 0], [9E9, 9E9, 9E9, 9E9, 9E9, 9E9]];
    CONST robtarget p16513:= [[1512.5020332002334, -66.37224427224653, 1008.500033578516], [0, 0, 1, 0], [0, 0, 0, 0], [9E9, 9E9, 9E9, 9E9, 9E9, 9E9]];
    CONST robtarget p16514:= [[1512.2960386592251, -66.40935731412112, 1008.500033578516], [0, 0, 1, 0], [0, 0, 0, 0], [9E9, 9E9, 9E9, 9E9, 9E9, 9E9]];
    CONST robtarget p16515:= [[1511.07524051963, -66.66015452512531, 1008.500033578516], [0, 0, 1, 0], [0, 0, 0, 0], [9E9, 9E9, 9E9, 9E9, 9E9, 9E9]];
    CONST robtarget p16516:= [[1510.7607766464141, -66.70532906970263, 1008.500033578516], [0, 0, 1, 0], [0, 0, 0, 0], [9E9, 9E9, 9E9, 9E9, 9E9, 9E9]];
    CONST robtarget p16517:= [[1510.4576579464385, -66.73438134131075, 1008.500033578516], [0, 0, 1, 0], [0, 0, 0, 0], [9E9, 9E9, 9E9, 9E9, 9E9, 9E9]];
    CONST robtarget p16518:= [[1509.175525449168, -66.92323694010081, 1008.500033578516], [0, 0, 1, 0], [0, 0, 0, 0], [9E9, 9E9, 9E9, 9E9, 9E9, 9E9]];
    CONST robtarget p16519:= [[1508.8704251307008, -66.9726340302731, 1008.500033578516], [0, 0, 1, 0], [0, 0, 0, 0], [9E9, 9E9, 9E9, 9E9, 9E9, 9E9]];
    CONST robtarget p16520:= [[1508.5274592133258, -67.00288674607833, 1008.500033578516], [0, 0, 1, 0], [0, 0, 0, 0], [9E9, 9E9, 9E9, 9E9, 9E9, 9E9]];
    CONST robtarget p16521:= [[1508.0968348541699, -67.06769352778105, 1008.500033578516], [0, 0, 1, 0], [0, 0, 0, 0], [9E9, 9E9, 9E9, 9E9, 9E9, 9E9]];
    CONST robtarget p16522:= [[1508.0090563037545, -67.06607693541001, 1008.500033578516], [0, 0, 1, 0], [0, 0, 0, 0], [9E9, 9E9, 9E9, 9E9, 9E9, 9E9]];
    CONST robtarget p16523:= [[1506.6807744034338, -67.21331099397379, 1008.500033578516], [0, 0, 1, 0], [0, 0, 0, 0], [9E9, 9E9, 9E9, 9E9, 9E9, 9E9]];
    CONST robtarget p16524:= [[1505.809088268359, -67.31317034555462, 1008.500033578516], [0, 0, 1, 0], [0, 0, 0, 0], [9E9, 9E9, 9E9, 9E9, 9E9, 9E9]];
    CONST robtarget p16525:= [[1505.6188516743464, -67.34205454790835, 1008.500033578516], [0, 0, 1, 0], [0, 0, 0, 0], [9E9, 9E9, 9E9, 9E9, 9E9, 9E9]];
    CONST robtarget p16526:= [[1504.8644377490357, -67.39601870094432, 1008.500033578516], [0, 0, 1, 0], [0, 0, 0, 0], [9E9, 9E9, 9E9, 9E9, 9E9, 9E9]];
    CONST robtarget p16527:= [[1504.407235656057, -67.42212820343448, 1008.500033578516], [0, 0, 1, 0], [0, 0, 0, 0], [9E9, 9E9, 9E9, 9E9, 9E9, 9E9]];
    CONST robtarget p16528:= [[1504.1697619267766, -67.44257116832785, 1008.500033578516], [0, 0, 1, 0], [0, 0, 0, 0], [9E9, 9E9, 9E9, 9E9, 9E9, 9E9]];
    CONST robtarget p16529:= [[1503.8256727741543, -67.46081649414805, 1008.500033578516], [0, 0, 1, 0], [0, 0, 0, 0], [9E9, 9E9, 9E9, 9E9, 9E9, 9E9]];
    CONST robtarget p16530:= [[1503.190405970635, -67.51523789385305, 1008.500033578516], [0, 0, 1, 0], [0, 0, 0, 0], [9E9, 9E9, 9E9, 9E9, 9E9, 9E9]];
    CONST robtarget p16531:= [[1502.9568800834174, -67.54164379967814, 1008.500033578516], [0, 0, 1, 0], [0, 0, 0, 0], [9E9, 9E9, 9E9, 9E9, 9E9, 9E9]];
    CONST robtarget p16532:= [[1502.5546042126823, -67.55982894154151, 1008.500033578516], [0, 0, 1, 0], [0, 0, 0, 0], [9E9, 9E9, 9E9, 9E9, 9E9, 9E9]];
    CONST robtarget p16533:= [[1502.0686149782923, -67.56494771918898, 1008.500033578516], [0, 0, 1, 0], [0, 0, 0, 0], [9E9, 9E9, 9E9, 9E9, 9E9, 9E9]];
    CONST robtarget p16534:= [[1500.8758617295618, -67.55694361813427, 1008.500033578516], [0, 0, 1, 0], [0, 0, 0, 0], [9E9, 9E9, 9E9, 9E9, 9E9, 9E9]];
    CONST robtarget p16535:= [[1500.565328073474, -67.54982645117659, 1008.500033578516], [0, 0, 1, 0], [0, 0, 0, 0], [9E9, 9E9, 9E9, 9E9, 9E9, 9E9]];
    CONST robtarget p16536:= [[1499.7668015366942, -67.50245784166341, 1008.500033578516], [0, 0, 1, 0], [0, 0, 0, 0], [9E9, 9E9, 9E9, 9E9, 9E9, 9E9]];
    CONST robtarget p16537:= [[1499.0308685030354, -67.52896885077217, 1008.500033578516], [0, 0, 1, 0], [0, 0, 0, 0], [9E9, 9E9, 9E9, 9E9, 9E9, 9E9]];
    CONST robtarget p16538:= [[1498.7722418163369, -67.5465495383315, 1008.500033578516], [0, 0, 1, 0], [0, 0, 0, 0], [9E9, 9E9, 9E9, 9E9, 9E9, 9E9]];
    CONST robtarget p16539:= [[1498.4191712373408, -67.56863004301617, 1008.500033578516], [0, 0, 1, 0], [0, 0, 0, 0], [9E9, 9E9, 9E9, 9E9, 9E9, 9E9]];
    CONST robtarget p16540:= [[1498.1829931551613, -67.56894347405097, 1008.500033578516], [0, 0, 1, 0], [0, 0, 0, 0], [9E9, 9E9, 9E9, 9E9, 9E9, 9E9]];
    CONST robtarget p16541:= [[1498.0600871550305, -67.5599913695027, 1008.500033578516], [0, 0, 1, 0], [0, 0, 0, 0], [9E9, 9E9, 9E9, 9E9, 9E9, 9E9]];
    CONST robtarget p16542:= [[1497.8860847948815, -67.5497451099145, 1008.500033578516], [0, 0, 1, 0], [0, 0, 0, 0], [9E9, 9E9, 9E9, 9E9, 9E9, 9E9]];
    CONST robtarget p16543:= [[1497.083111233579, -67.53643456396763, 1008.500033578516], [0, 0, 1, 0], [0, 0, 0, 0], [9E9, 9E9, 9E9, 9E9, 9E9, 9E9]];
    CONST robtarget p16544:= [[1496.4314673256445, -67.47528980158458, 1008.500033578516], [0, 0, 1, 0], [0, 0, 0, 0], [9E9, 9E9, 9E9, 9E9, 9E9, 9E9]];
    CONST robtarget p16545:= [[1496.3198801716283, -67.46968728757439, 1008.500033578516], [0, 0, 1, 0], [0, 0, 0, 0], [9E9, 9E9, 9E9, 9E9, 9E9, 9E9]];
    CONST robtarget p16546:= [[1495.8621445522426, -67.45416099025189, 1008.500033578516], [0, 0, 1, 0], [0, 0, 0, 0], [9E9, 9E9, 9E9, 9E9, 9E9, 9E9]];
    CONST robtarget p16547:= [[1494.989762580834, -67.38331726780963, 1008.500033578516], [0, 0, 1, 0], [0, 0, 0, 0], [9E9, 9E9, 9E9, 9E9, 9E9, 9E9]];
    CONST robtarget p16548:= [[1494.4087875372004, -67.34314190342765, 1008.500033578516], [0, 0, 1, 0], [0, 0, 0, 0], [9E9, 9E9, 9E9, 9E9, 9E9, 9E9]];
    CONST robtarget p16549:= [[1494.0247160945187, -67.31910795155888, 1008.500033578516], [0, 0, 1, 0], [0, 0, 0, 0], [9E9, 9E9, 9E9, 9E9, 9E9, 9E9]];
    CONST robtarget p16550:= [[1493.5917069247707, -67.28956139083931, 1008.500033578516], [0, 0, 1, 0], [0, 0, 0, 0], [9E9, 9E9, 9E9, 9E9, 9E9, 9E9]];
    CONST robtarget p16551:= [[1492.9653848149794, -67.2397719487922, 1008.500033578516], [0, 0, 1, 0], [0, 0, 0, 0], [9E9, 9E9, 9E9, 9E9, 9E9, 9E9]];
    CONST robtarget p16552:= [[1492.6590504024691, -67.1861070504822, 1008.500033578516], [0, 0, 1, 0], [0, 0, 0, 0], [9E9, 9E9, 9E9, 9E9, 9E9, 9E9]];
    CONST robtarget p16553:= [[1492.1668974353709, -67.0997183976802, 1008.500033578516], [0, 0, 1, 0], [0, 0, 0, 0], [9E9, 9E9, 9E9, 9E9, 9E9, 9E9]];
    CONST robtarget p16554:= [[1492.0157173001858, -67.06845223036602, 1008.500033578516], [0, 0, 1, 0], [0, 0, 0, 0], [9E9, 9E9, 9E9, 9E9, 9E9, 9E9]];
    CONST robtarget p16555:= [[1491.3440320613395, -66.98013332050493, 1008.500033578516], [0, 0, 1, 0], [0, 0, 0, 0], [9E9, 9E9, 9E9, 9E9, 9E9, 9E9]];
    CONST robtarget p16556:= [[1491.0305381525786, -66.96721071543787, 1008.500033578516], [0, 0, 1, 0], [0, 0, 0, 0], [9E9, 9E9, 9E9, 9E9, 9E9, 9E9]];
    CONST robtarget p16557:= [[1490.6190875430814, -66.91541707324892, 1008.500033578516], [0, 0, 1, 0], [0, 0, 0, 0], [9E9, 9E9, 9E9, 9E9, 9E9, 9E9]];
    CONST robtarget p16558:= [[1490.017914883082, -66.8017127111406, 1008.500033578516], [0, 0, 1, 0], [0, 0, 0, 0], [9E9, 9E9, 9E9, 9E9, 9E9, 9E9]];
    CONST robtarget p16559:= [[1489.6833658314138, -66.76514251421887, 1008.500033578516], [0, 0, 1, 0], [0, 0, 0, 0], [9E9, 9E9, 9E9, 9E9, 9E9, 9E9]];
    CONST robtarget p16560:= [[1488.9923903907588, -66.67249914822163, 1008.500033578516], [0, 0, 1, 0], [0, 0, 0, 0], [9E9, 9E9, 9E9, 9E9, 9E9, 9E9]];
    CONST robtarget p16561:= [[1488.8420142559903, -66.66158025702326, 1008.500033578516], [0, 0, 1, 0], [0, 0, 0, 0], [9E9, 9E9, 9E9, 9E9, 9E9, 9E9]];
    CONST robtarget p16562:= [[1488.191627629811, -66.56893860366978, 1008.500033578516], [0, 0, 1, 0], [0, 0, 0, 0], [9E9, 9E9, 9E9, 9E9, 9E9, 9E9]];
    CONST robtarget p16563:= [[1487.6804547151357, -66.4685656525345, 1008.500033578516], [0, 0, 1, 0], [0, 0, 0, 0], [9E9, 9E9, 9E9, 9E9, 9E9, 9E9]];
    CONST robtarget p16564:= [[1487.0055162106032, -66.33810741666336, 1008.500033578516], [0, 0, 1, 0], [0, 0, 0, 0], [9E9, 9E9, 9E9, 9E9, 9E9, 9E9]];
    CONST robtarget p16565:= [[1486.7975136269433, -66.28865723994846, 1008.500033578516], [0, 0, 1, 0], [0, 0, 0, 0], [9E9, 9E9, 9E9, 9E9, 9E9, 9E9]];
    CONST robtarget p16566:= [[1486.5735170616765, -66.21605235557095, 1008.500033578516], [0, 0, 1, 0], [0, 0, 0, 0], [9E9, 9E9, 9E9, 9E9, 9E9, 9E9]];
    CONST robtarget p16567:= [[1486.08334772369, -66.06780085596483, 1008.500033578516], [0, 0, 1, 0], [0, 0, 0, 0], [9E9, 9E9, 9E9, 9E9, 9E9, 9E9]];
    CONST robtarget p16568:= [[1484.8724515212464, -65.85857803760453, 1008.500033578516], [0, 0, 1, 0], [0, 0, 0, 0], [9E9, 9E9, 9E9, 9E9, 9E9, 9E9]];
    CONST robtarget p16569:= [[1484.813178416727, -65.84258766832549, 1008.500033578516], [0, 0, 1, 0], [0, 0, 0, 0], [9E9, 9E9, 9E9, 9E9, 9E9, 9E9]];
    CONST robtarget p16570:= [[1484.1561133766663, -65.69798811455867, 1008.500033578516], [0, 0, 1, 0], [0, 0, 0, 0], [9E9, 9E9, 9E9, 9E9, 9E9, 9E9]];
    CONST robtarget p16571:= [[1483.957584377456, -65.65404041841009, 1008.500033578516], [0, 0, 1, 0], [0, 0, 0, 0], [9E9, 9E9, 9E9, 9E9, 9E9, 9E9]];
    CONST robtarget p16572:= [[1482.9422162637081, -65.42671662294471, 1008.500033578516], [0, 0, 1, 0], [0, 0, 0, 0], [9E9, 9E9, 9E9, 9E9, 9E9, 9E9]];
    CONST robtarget p16573:= [[1482.6347655776838, -65.31356696231464, 1008.500033578516], [0, 0, 1, 0], [0, 0, 0, 0], [9E9, 9E9, 9E9, 9E9, 9E9, 9E9]];
    CONST robtarget p16574:= [[1482.3180616266495, -65.21608131509697, 1008.500033578516], [0, 0, 1, 0], [0, 0, 0, 0], [9E9, 9E9, 9E9, 9E9, 9E9, 9E9]];
    CONST robtarget p16575:= [[1481.975400777133, -65.13348433134436, 1008.500033578516], [0, 0, 1, 0], [0, 0, 0, 0], [9E9, 9E9, 9E9, 9E9, 9E9, 9E9]];
    CONST robtarget p16576:= [[1481.6807117175858, -65.03478079956349, 1008.500033578516], [0, 0, 1, 0], [0, 0, 0, 0], [9E9, 9E9, 9E9, 9E9, 9E9, 9E9]];
    CONST robtarget p16577:= [[1481.362285170357, -64.93940031305225, 1008.500033578516], [0, 0, 1, 0], [0, 0, 0, 0], [9E9, 9E9, 9E9, 9E9, 9E9, 9E9]];
    CONST robtarget p16578:= [[1480.4887824065574, -64.68796353048609, 1008.500033578516], [0, 0, 1, 0], [0, 0, 0, 0], [9E9, 9E9, 9E9, 9E9, 9E9, 9E9]];
    CONST robtarget p16579:= [[1480.378818998745, -64.65282237173975, 1008.500033578516], [0, 0, 1, 0], [0, 0, 0, 0], [9E9, 9E9, 9E9, 9E9, 9E9, 9E9]];
    CONST robtarget p16580:= [[1480.0514162015609, -64.552918643896, 1008.500033578516], [0, 0, 1, 0], [0, 0, 0, 0], [9E9, 9E9, 9E9, 9E9, 9E9, 9E9]];
    CONST robtarget p16581:= [[1479.7673149044228, -64.48115794995756, 1008.500033578516], [0, 0, 1, 0], [0, 0, 0, 0], [9E9, 9E9, 9E9, 9E9, 9E9, 9E9]];
    CONST robtarget p16582:= [[1478.8558026242943, -64.17858766362941, 1008.500033578516], [0, 0, 1, 0], [0, 0, 0, 0], [9E9, 9E9, 9E9, 9E9, 9E9, 9E9]];
    CONST robtarget p16583:= [[1478.5196895925658, -64.07092275092666, 1008.500033578516], [0, 0, 1, 0], [0, 0, 0, 0], [9E9, 9E9, 9E9, 9E9, 9E9, 9E9]];
    CONST robtarget p16584:= [[1477.7438998468722, -63.837843656361095, 1008.500033578516], [0, 0, 1, 0], [0, 0, 0, 0], [9E9, 9E9, 9E9, 9E9, 9E9, 9E9]];
    CONST robtarget p16585:= [[1477.3660620165274, -63.67014790234987, 1008.500033578516], [0, 0, 1, 0], [0, 0, 0, 0], [9E9, 9E9, 9E9, 9E9, 9E9, 9E9]];
    CONST robtarget p16586:= [[1477.0588507031564, -63.51673046398417, 1008.500033578516], [0, 0, 1, 0], [0, 0, 0, 0], [9E9, 9E9, 9E9, 9E9, 9E9, 9E9]];
    CONST robtarget p16587:= [[1475.9738168880424, -63.16147628801768, 1008.500033578516], [0, 0, 1, 0], [0, 0, 0, 0], [9E9, 9E9, 9E9, 9E9, 9E9, 9E9]];
    CONST robtarget p16588:= [[1475.6713805261898, -63.0439147743457, 1008.500033578516], [0, 0, 1, 0], [0, 0, 0, 0], [9E9, 9E9, 9E9, 9E9, 9E9, 9E9]];
    CONST robtarget p16589:= [[1475.1812018381816, -62.84947227434736, 1008.500033578516], [0, 0, 1, 0], [0, 0, 0, 0], [9E9, 9E9, 9E9, 9E9, 9E9, 9E9]];
    CONST robtarget p16590:= [[1474.7614695275313, -62.693750639007646, 1008.500033578516], [0, 0, 1, 0], [0, 0, 0, 0], [9E9, 9E9, 9E9, 9E9, 9E9, 9E9]];
    CONST robtarget p16591:= [[1474.16884731843, -62.46002910612246, 1008.500033578516], [0, 0, 1, 0], [0, 0, 0, 0], [9E9, 9E9, 9E9, 9E9, 9E9, 9E9]];
    CONST robtarget p16592:= [[1473.8649397416566, -62.34261433569378, 1008.500033578516], [0, 0, 1, 0], [0, 0, 0, 0], [9E9, 9E9, 9E9, 9E9, 9E9, 9E9]];
    CONST robtarget p16593:= [[1472.6352606001096, -61.784068147206455, 1008.500033578516], [0, 0, 1, 0], [0, 0, 0, 0], [9E9, 9E9, 9E9, 9E9, 9E9, 9E9]];
    CONST robtarget p16594:= [[1471.8701483786922, -61.362740064126285, 1008.500033578516], [0, 0, 1, 0], [0, 0, 0, 0], [9E9, 9E9, 9E9, 9E9, 9E9, 9E9]];
    CONST robtarget p16595:= [[1471.412616980215, -61.16760242585946, 1008.500033578516], [0, 0, 1, 0], [0, 0, 0, 0], [9E9, 9E9, 9E9, 9E9, 9E9, 9E9]];
    CONST robtarget p16596:= [[1470.7539359434206, -60.895908701576076, 1008.500033578516], [0, 0, 1, 0], [0, 0, 0, 0], [9E9, 9E9, 9E9, 9E9, 9E9, 9E9]];
    CONST robtarget p16597:= [[1470.3108003811822, -60.68318012989036, 1008.500033578516], [0, 0, 1, 0], [0, 0, 0, 0], [9E9, 9E9, 9E9, 9E9, 9E9, 9E9]];
    CONST robtarget p16598:= [[1470.1695883225386, -60.60870884877002, 1008.500033578516], [0, 0, 1, 0], [0, 0, 0, 0], [9E9, 9E9, 9E9, 9E9, 9E9, 9E9]];
    CONST robtarget p16599:= [[1469.584722450983, -60.330203876399246, 1008.500033578516], [0, 0, 1, 0], [0, 0, 0, 0], [9E9, 9E9, 9E9, 9E9, 9E9, 9E9]];
    CONST robtarget p16600:= [[1468.8297289676302, -59.93336743589276, 1008.500033578516], [0, 0, 1, 0], [0, 0, 0, 0], [9E9, 9E9, 9E9, 9E9, 9E9, 9E9]];
    CONST robtarget p16601:= [[1468.5525163101865, -59.77330352083022, 1008.500033578516], [0, 0, 1, 0], [0, 0, 0, 0], [9E9, 9E9, 9E9, 9E9, 9E9, 9E9]];
    CONST robtarget p16602:= [[1468.3542149028913, -59.66020211090191, 1008.500033578516], [0, 0, 1, 0], [0, 0, 0, 0], [9E9, 9E9, 9E9, 9E9, 9E9, 9E9]];
    CONST robtarget p16603:= [[1468.0476624993591, -59.50108991428728, 1008.500033578516], [0, 0, 1, 0], [0, 0, 0, 0], [9E9, 9E9, 9E9, 9E9, 9E9, 9E9]];
    CONST robtarget p16604:= [[1467.260552521564, -59.08985536104261, 1008.500033578516], [0, 0, 1, 0], [0, 0, 0, 0], [9E9, 9E9, 9E9, 9E9, 9E9, 9E9]];
    CONST robtarget p16605:= [[1466.2732364950225, -58.548428748402976, 1008.500033578516], [0, 0, 1, 0], [0, 0, 0, 0], [9E9, 9E9, 9E9, 9E9, 9E9, 9E9]];
    CONST robtarget p16606:= [[1465.7181347981434, -58.22140113027264, 1008.500033578516], [0, 0, 1, 0], [0, 0, 0, 0], [9E9, 9E9, 9E9, 9E9, 9E9, 9E9]];
    CONST robtarget p16607:= [[1465.3010168289268, -58.01426917306288, 1008.500033578516], [0, 0, 1, 0], [0, 0, 0, 0], [9E9, 9E9, 9E9, 9E9, 9E9, 9E9]];
    CONST robtarget p16608:= [[1464.916394542098, -57.75543720706439, 1008.500033578516], [0, 0, 1, 0], [0, 0, 0, 0], [9E9, 9E9, 9E9, 9E9, 9E9, 9E9]];
    CONST robtarget p16609:= [[1464.3430536964283, -57.43295207521634, 1008.500033578516], [0, 0, 1, 0], [0, 0, 0, 0], [9E9, 9E9, 9E9, 9E9, 9E9, 9E9]];
    CONST robtarget p16610:= [[1464.2432213462987, -57.37253118745075, 1008.500033578516], [0, 0, 1, 0], [0, 0, 0, 0], [9E9, 9E9, 9E9, 9E9, 9E9, 9E9]];
    CONST robtarget p16611:= [[1463.8731514613346, -57.08630293884973, 1008.500033578516], [0, 0, 1, 0], [0, 0, 0, 0], [9E9, 9E9, 9E9, 9E9, 9E9, 9E9]];
    CONST robtarget p16612:= [[1463.6300861065854, -56.92584405997732, 1008.500033578516], [0, 0, 1, 0], [0, 0, 0, 0], [9E9, 9E9, 9E9, 9E9, 9E9, 9E9]];
    CONST robtarget p16613:= [[1463.17392362813, -56.65701374013654, 1008.500033578516], [0, 0, 1, 0], [0, 0, 0, 0], [9E9, 9E9, 9E9, 9E9, 9E9, 9E9]];
    CONST robtarget p16614:= [[1463.106287518344, -56.60777995069512, 1008.500033578516], [0, 0, 1, 0], [0, 0, 0, 0], [9E9, 9E9, 9E9, 9E9, 9E9, 9E9]];
    CONST robtarget p16615:= [[1462.5604227603878, -56.23990891753269, 1008.500033578516], [0, 0, 1, 0], [0, 0, 0, 0], [9E9, 9E9, 9E9, 9E9, 9E9, 9E9]];
    CONST robtarget p16616:= [[1462.118208957654, -55.934225856163664, 1008.500033578516], [0, 0, 1, 0], [0, 0, 0, 0], [9E9, 9E9, 9E9, 9E9, 9E9, 9E9]];
    CONST robtarget p16617:= [[1461.877608039019, -55.78661021882508, 1008.500033578516], [0, 0, 1, 0], [0, 0, 0, 0], [9E9, 9E9, 9E9, 9E9, 9E9, 9E9]];
    CONST robtarget p16618:= [[1461.6943555925486, -55.684046011661835, 1008.500033578516], [0, 0, 1, 0], [0, 0, 0, 0], [9E9, 9E9, 9E9, 9E9, 9E9, 9E9]];
